(* IEC 61131-3 sources: elnaProjects/ElpcLogic/PomarKc7Changed/FunctionBlocks (part 6) *)

(* ---- ppuAlg.st ---- *)
FUNCTION_BLOCK ppuAlg

VAR_IN_OUT
	StrAlg : struct_Alg;
END_VAR

VAR
	BMP_Err : struct_PhaseAlgoritm;
	Level_masla_Norm : struct_PhaseAlgoritm;
	T_masla_Norm : struct_PhaseAlgoritm;
	Krans_ready_to_move : struct_PhaseAlgoritm;
END_VAR

VAR_IN_OUT
	Krans_Poloj : struct_PhaseAlgoritm;
	Net_AO_KC_SHKS04M : struct_PhaseAlgoritm;
	EGPA_Stop : struct_PhaseAlgoritm;
	Avt_SHU_vkl : struct_PhaseAlgoritm;
	All_IM_Off : struct_PhaseAlgoritm;
	Nalichie220_SHU_Ai : struct_PhaseAlgoritm;
	BP_Norm : struct_PhaseAlgoritm;
	Naprajenie_U_IM : struct_PhaseAlgoritm;
	MV_Poloj_RolledON : struct_PhaseAlgoritm;
	MV_Poloj_RolledOFF : struct_PhaseAlgoritm;
	NOTAnalogNS : struct_PhaseAlgoritm;
	Net_ASPS_Analogs : struct_PhaseAlgoritm;
	Not_AS : struct_PhaseAlgoritm;
	Gotov_Vozb : struct_PhaseAlgoritm;
	Reactornyi_P : struct_PhaseAlgoritm;
	Chastotnyi_P : struct_PhaseAlgoritm;
	dP_kr1 : struct_PhaseAlgoritm;
	Auto_Rej : struct_PhaseAlgoritm;
	CK_IM_Norm : struct_PhaseAlgoritm;
	HAnd_Mode : struct_PhaseAlgoritm;
	Impuls_Gaz : struct_PhaseAlgoritm;
END_VAR

VAR
	fb_BMP_Err : fb_ph_CustomPhase;
	fb_Level_masla_Norm : fb_ph_CustomPhase;
	fb_T_masla_Norm : fb_ph_CustomPhase;
	fb_Krans_ready_to_move : fb_ph_CustomPhase;
	fb_Krans_Poloj : fb_ph_CustomPhase;
	fb_Net_AO_KC_SHKS04M : fb_ph_CustomPhase;
	fb_EGPA_Stop : fb_ph_CustomPhase;
	fb_Avt_SHU_vkl : fb_ph_CustomPhase;
	fb_All_IM_Off : fb_ph_CustomPhase;
	fb_Nalichie220_SHU_Ai : fb_ph_CustomPhase;
	fb_BP_Norm : fb_ph_CustomPhase;
	fb_Naprajenie_U_IM : fb_ph_CustomPhase;
	fb_MV_Poloj_RolledON : fb_ph_CustomPhase;
	fb_MV_Poloj_RolledOFF : fb_ph_CustomPhase;
	fb_NOTAnalogNS : fb_ph_CustomPhase;
	fb_Net_ASPS_Analogs : fb_ph_CustomPhase;
	fb_Not_AS : fb_ph_CustomPhase;
	fb_Gotov_Vozb : fb_ph_CustomPhase;
	fb_Reactornyi_P : fb_ph_CustomPhase;
	fb_Chastotnyi_P : fb_ph_CustomPhase;
	fb_dP_kr1 : fb_ph_CustomPhase;
	fb_Auto_Rej : fb_ph_CustomPhase;
	fb_CK_IM_Norm : fb_ph_CustomPhase;
	fb_HAnd_Mode : fb_ph_CustomPhase;
	fb_Impuls_Gaz : fb_ph_CustomPhase;
	_sunpackerCommand : fb_sunpackerCommand;
	modeR_Trig : R_TRIG;
	modeF_Trig : F_TRIG;
	_statusAi : TYPE_StatusAi;
	_Answers : TYPE_Answers;
	_statusDualInput : TYPE_statusDualInput;
	_DualStateImAction : TYPE_DualStateImAction;
	_PhaseAlgoritmAction : TYPE_PhaseAlgoritmAction;
	_basketStats : TYPE_basketStats;
END_VAR

VAR_OUTPUT
	puskAllowed : BOOL;
	testAllowed : BOOL;
END_VAR

VAR
	ppuDone : BOOL;
	source : BYTE;
	cmd : BYTE;
	lastCmd : BYTE;
	source_for_Status : BYTE;
	cmd_for_Status : BYTE;
	command_error_for_Status : BYTE;
	resetCmdTimer : TON;
	resetCmdTimerPriznak : BOOL;
	onInit : BOOL;
END_VAR

VAR_EXTERNAL
	IM : ImConfig;
	ai : AiConfig;
	di : DiConfig;
	algManager : struct_AlgoritmsManager;
	protectManager : struct_ProtectionsManager;
	NotHasRezervNU : BOOL;
	ModeGpa : TYPE_ModeGpa;
	algoritms : AlgoritmsConfig;
END_VAR

IF NOT onInit THEN

    fb_BMP_Err(phaseNumber:=0);
    fb_Level_masla_Norm(phaseNumber:=1);
    fb_T_masla_Norm(phaseNumber:=2);
    fb_Krans_ready_to_move(phaseNumber:=5);
    fb_Krans_Poloj(phaseNumber:=6);
    fb_Net_AO_KC_SHKS04M(phaseNumber:=7);
    fb_EGPA_Stop(phaseNumber:=9);
    fb_Avt_SHU_vkl(phaseNumber:=10);
    fb_All_IM_Off(phaseNumber:=11);
    fb_Nalichie220_SHU_Ai(phaseNumber:=12);
    fb_BP_Norm(phaseNumber:=13);
    fb_Naprajenie_U_IM(phaseNumber:=14);
    fb_MV_Poloj_RolledON(phaseNumber:=15);
    fb_MV_Poloj_RolledOFF(phaseNumber:=16);
    fb_NOTAnalogNS(phaseNumber:=17);
    fb_Net_ASPS_Analogs(phaseNumber:=18);
    fb_Not_AS(phaseNumber:=19);
    fb_Gotov_Vozb(phaseNumber:=20);
    fb_Reactornyi_P(phaseNumber:=21);
    fb_Chastotnyi_P(phaseNumber:=22);
    fb_dP_kr1(phaseNumber:=23);
    fb_Auto_Rej(phaseNumber:=24);
    fb_CK_IM_Norm(phaseNumber:=25);
    fb_HAnd_Mode(phaseNumber:=26);
    fb_Impuls_Gaz(phaseNumber:=27);

onInit:=TRUE;
END_IF;

fb_BMP_Err(StrPh:=BMP_Err);
fb_Level_masla_Norm(StrPh:=Level_masla_Norm);
fb_T_masla_Norm(StrPh:=T_masla_Norm);
fb_Krans_ready_to_move(StrPh:=Krans_ready_to_move);
fb_Krans_Poloj(StrPh:=Krans_Poloj);
fb_Net_AO_KC_SHKS04M(StrPh:=Net_AO_KC_SHKS04M);
fb_EGPA_Stop(StrPh:=EGPA_Stop);
fb_Avt_SHU_vkl(StrPh:=Avt_SHU_vkl);
fb_All_IM_Off(StrPh:=All_IM_Off);
fb_Nalichie220_SHU_Ai(StrPh:=Nalichie220_SHU_Ai);
fb_BP_Norm(StrPh:=BP_Norm);
fb_Naprajenie_U_IM(StrPh:=Naprajenie_U_IM);
fb_MV_Poloj_RolledON(StrPh:=MV_Poloj_RolledON);
fb_MV_Poloj_RolledOFF(StrPh:=MV_Poloj_RolledOFF);
fb_NOTAnalogNS(StrPh:=NOTAnalogNS);
fb_Net_ASPS_Analogs(StrPh:=Net_ASPS_Analogs);
fb_Not_AS(StrPh:=Not_AS);
fb_Gotov_Vozb(StrPh:=Gotov_Vozb);
fb_Reactornyi_P(StrPh:=Reactornyi_P);
fb_Chastotnyi_P(StrPh:=Chastotnyi_P);
fb_dP_kr1(StrPh:=dP_kr1);
fb_Auto_Rej(StrPh:=Auto_Rej);
fb_CK_IM_Norm(StrPh:=CK_IM_Norm);
fb_HAnd_Mode(StrPh:=HAnd_Mode);
fb_Impuls_Gaz(StrPh:=Impuls_Gaz);

IF StrAlg.isRuning THEN

    (*BMP_Err.top:= ((BMPERR_k = 0) OR (kontroller.imit)); надо разобраться кто такой BMPERR_k*)
    (*уровень масла в норме*)
    Level_masla_Norm.top := (ai.Yroven_masla_MB.interval = _statusAi.normal);

    (*температура масла в норме*)
    T_masla_Norm.top:= (ai.Tmasla_MB.interval = _statusAi.normal);

    (*kраны готовы к управлению*)
    Krans_ready_to_move.top:= NOT (IM.Kran1.So OR IM.Kran1.Sz OR IM.Kran2.So OR IM.Kran2.Sz OR IM.Kran3.So OR
                                   IM.Kran3.Sz OR IM.Kran3b.So OR IM.Kran3b.Sz OR IM.Kran4.So OR IM.Kran4.Sz OR
			     IM.Kran5.So OR IM.Kran5.Sz OR IM.Kran6.So OR IM.Kran6.Sz);

    (*положение кранов верное*)
    Krans_Poloj.top:= (Im.Kran1.onStatus=_statusDualInput.STATUS_OFF) AND
		  (Im.Kran2.onStatus=_statusDualInput.STATUS_OFF) AND
		  (Im.Kran3.onStatus=_statusDualInput.STATUS_OFF) AND
		  (Im.Kran3b.onStatus=_statusDualInput.STATUS_ON) AND
		  (Im.Kran4.onStatus=_statusDualInput.STATUS_OFF) AND
		  (Im.Kran5.onStatus=_statusDualInput.STATUS_ON) AND
                      (Im.Kran6.onStatus=_statusDualInput.STATUS_ON);
    (*Нет АО от ШКС
    Net_AO_KC_SHKS04M.top:= haveAlarms(); кто такой haveAlarms*)

    (*Режим ЭГПА остановлен *)
    EGPA_Stop.top := (algManager.mode = ModeGpa.MODE_STOP);

    (*Автомат ШУ включен *)
    Avt_SHU_vkl.top := IM.SingleSignals.SHU_v_GPA_vkluch.Q;

    (*Все исполнительные механизмы выключены *)
    All_IM_Off.top := (IM.mv.onStatus=_statusDualInput.STATUS_OFF) AND (IM.pns.onStatus=_statusDualInput.STATUS_OFF) AND
                      (IM.nu1.onStatus=_statusDualInput.STATUS_OFF) AND (IM.nu2.onStatus=_statusDualInput.STATUS_OFF) AND
                      (IM.v1_Avom.onStatus=_statusDualInput.STATUS_OFF) AND (IM.v2_Avom.onStatus=_statusDualInput.STATUS_OFF) AND
		  (IM.v3_Avom.onStatus=_statusDualInput.STATUS_OFF)AND (IM.v4_Avom.onStatus=_statusDualInput.STATUS_OFF) AND
                      (IM.CMN.onStatus=_statusDualInput.STATUS_OFF) AND (IM.TEN_MB.onStatus=_statusDualInput.STATUS_OFF) AND
                      (IM.TEN_kollectora.onStatus=_statusDualInput.STATUS_OFF) AND (IM.KaloriferAVOM.onStatus=_statusDualInput.STATUS_OFF);

    (*Наличие 220 в шу*)
    Nalichie220_SHU_Ai.top :=	(ai.Kontrol_per_220V.interval = _statusAi.normal)	 AND (ai.Kontrol_post_220V.interval = _statusAi.normal);

    (*Блоки питания норм*)
    BP_Norm.top:=
		(IM.SingleSignals.Nalichie_BP1.Q AND
		IM.SingleSignals.Nalichie_BP2.Q AND
		IM.SingleSignals.Nalichie_BP3.Q AND
		IM.SingleSignals.Nalichie_BP4.Q AND
		IM.SingleSignals.Nalichie_BP5.Q AND
		IM.SingleSignals.Nalichie_BP6.Q AND
		IM.SingleSignals.Nalichie_BP7_BP8.Q AND
		IM.SingleSignals.Nalichie_BP9_BP10.Q AND

		IM.SingleSignals.Nalichie_220BEAO.Q AND
		IM.SingleSignals.Nalichie_per_220_na_vhode.Q AND
		IM.SingleSignals.Nalichie_post_220_na_vhode.Q AND
		IM.SingleSignals.Nalichie_BP11.Q AND
		IM.SingleSignals.Nalichie_BP12.Q);

    (*Напряжение исполнительниых механизмов
    Naprajenie_U_IM.top := IM.NalichieU_CMN.q AND IM.NalichieU_NU1.Q AND IM.Nalichie_CU_MV.Q  AND IM.NalichieU_NU2.Q AND
						IM.NalichieU_PNS.Q; нет сигналов таких *)

    (* положение тележки мв вкачена *)
    MV_Poloj_RolledON.top:= IM.mv.basketStatus = _basketStats.BASKET_ROLLEDIN;

    (* положение тележки мв выкачена *)
    MV_Poloj_RolledOFF.top:= IM.mv.basketStatus = _basketStats.BASKET_ROLLEDOUT;

    (* нет неисправных аналоговых сигналов *)
    NOTAnalogNS.top :=  NOT analogsNS();

    (* нет аварийных/предупредительных сигнализаций аналоговых сигналов *)
    Net_ASPS_Analogs.top := anyAnalogsPs(); (*Не понял где посмотреть наличие ас аналогов *)

    (* нет сработанных защит *)
    Not_AS.top := NOT anyProtectionSignaling();

    (* готовность возбудителя *)
    Gotov_Vozb.top:= IM.SingleSignals.Vozbud_gotovnost.Q;

    (* реакторный пуск *)
    Reactornyi_P.top := IM.SingleSignals.Reactorny_pusk.Q AND NOT IM.SingleSignals.Chastotny_pusk.Q;

    (* частотный пуск *)
    Chastotnyi_P.top:=IM.SingleSignals.Chastotny_pusk.Q AND NOT IM.SingleSignals.Reactorny_pusk.Q;

    (* нет перепада давления на кране 1 *)
    dP_kr1.top:= NOT IM.SingleSignals.dp_kran1_Less100.Q (*AND (IM.PerepadDavlenieKran1_CK.status = 1))*);

    (* в автоматическом ли режиме исполнительные механизмы *)
    (*Auto_Rej.top := im.NU1_Automat.Q AND im.PNS_Automat.Q AND im.NU2_Automat.Q;*)

    (* есть наряжение в цепях управления ИМ *)
    CK_IM_Norm.top := nsCepeiUpravlenya();

    (* ручной режим *)
    HAnd_Mode.top:= NOT im.SingleSignals.Rezhim_ruchnogo_regulirovaniya.Q;

    (* импульсный газ *)
    Impuls_Gaz.top:= ai.Pimpuls_gaz.interval=_statusAi.normal;

    ppuDone := BMP_Err.top AND
	     Level_masla_Norm.top AND
               T_masla_Norm.top AND
	     Krans_ready_to_move.top AND
	     Krans_Poloj.top AND
	     Net_AO_KC_SHKS04M.top AND
	     EGPA_Stop.top AND
               Avt_SHU_vkl.top AND
               All_IM_Off.top AND
               Nalichie220_SHU_Ai.top AND
               BP_Norm.top AND
               Naprajenie_U_IM.top AND
               MV_Poloj_RolledON.top AND
               MV_Poloj_RolledOFF.top AND
               NOTAnalogNS.top AND
               Net_ASPS_Analogs.top AND
               Not_AS.top AND
               Gotov_Vozb.top AND
               Reactornyi_P.top AND
               Chastotnyi_P.top AND
               dP_kr1.top AND
               Auto_Rej.top AND
               CK_IM_Norm.top AND
               HAnd_Mode.top AND
               Impuls_Gaz.top;

    puskAllowed:= ppuDone AND Im.mv.basketStatus = _basketStats.BASKET_ROLLEDIN;
    testAllowed:= ppuDone AND Im.mv.basketStatus = _basketStats.BASKET_ROLLEDOUT;

    modeR_Trig(CLK:=puskAllowed);
    modeF_Trig(CLK:=puskAllowed);

    IF modeR_Trig.Q THEN
	algManager.nMode:= ModeGpa.MODE_READY;
    END_IF;
    IF modeF_Trig.Q THEN
	algManager.nMode:= ModeGpa.MODE_STOP;
    END_IF;

    IF puskAllowed THEN
        algoritms.Apusk.inCanRun:= TRUE;
        algoritms.SemiAutoPusk.inCanRun:= TRUE;
    ELSE
        algoritms.Apusk.inCanRun:= FALSE;
        algoritms.SemiAutoPusk.inCanRun:= FALSE;
    END_IF;

    IF testAllowed THEN
        algoritms.testPms.inCanRun:=  TRUE;
        algoritms.testdPmg.inCanRun:= TRUE;
        algoritms.puskK.inCanRun:=    TRUE;
        algoritms.puskV.inCanRun:=    TRUE;
    ELSE
        algoritms.testPms.inCanRun:=  FALSE;
        algoritms.testdPmg.inCanRun:= FALSE;
        algoritms.puskK.inCanRun:=    FALSE;
        algoritms.puskV.inCanRun:=    FALSE;
    END_IF;

END_IF;

StrAlg.CanRun := StrAlg.inCanRun;
StrAlg.OpcCommandsDisabled := StrAlg.inOpcCommandsDisabled;

(* ---- Если управление с ВУ заблокировано, то  передаем команду из алгоритма ---- *)
IF StrAlg.inOpcCommandsDisabled THEN
	StrAlg.inCommand := StrAlg.inCommand_Alg;
ELSE (* иначе передаем команду с АРМа*)
	StrAlg.inCommand := StrAlg.inCommand_ARM;
END_IF;

_sunpackerCommand(command := StrAlg.inCommand);
	source := _sunpackerCommand.source;
	cmd := _sunpackerCommand.cmd;

IF cmd <> 0 AND lastCmd <> cmd AND (((NOT StrAlg.opcCommandsDisabled) AND source > 0) OR source = 0) then
	CASE BYTE_TO_INT(cmd) OF
		(*cmdRun*) 1: 	IF (StrAlg.CanRun) THEN
					StrAlg.isRuning := TRUE;
					StrAlg.isEnded := FALSE;
					StrAlg.hasError := FALSE;
					(*****************       OnRun       *****************)

					cmd_for_Status := cmd;
					source_for_Status := source;
					command_error_for_Status := 0;
				ELSE
					StrAlg.isRuning := FALSE;
					StrAlg.isEnded := FALSE;
					StrAlg.hasError 	:= FALSE;

					cmd_for_Status := 0;
					source_for_Status := source;
					command_error_for_Status := cmd;
				END_IF;
		(*cmdReset*) 2: 	StrAlg.isRuning := FALSE;
				StrAlg.isEnded := FALSE;
				StrAlg.hasError 	:= FALSE;

                                         (*****************       OnReset       *****************)

                                                  resetPhase(BMP_Err);
                                                  resetPhase(Level_masla_Norm);
                                                  resetPhase(T_masla_Norm);
                                                  resetPhase(Krans_ready_to_move);
                                                  resetPhase(Krans_Poloj);
                                                  resetPhase(Net_AO_KC_SHKS04M);
                                                  resetPhase(EGPA_Stop);
                                                  resetPhase(Avt_SHU_vkl);
                                                  resetPhase(All_IM_Off);
                                                  resetPhase(Nalichie220_SHU_Ai);
                                                  resetPhase(BP_Norm);
                                                  resetPhase(Naprajenie_U_IM);
                                                  resetPhase(MV_Poloj_RolledON);
                                                  resetPhase(MV_Poloj_RolledOFF);
                                                  resetPhase(NOTAnalogNS);
                                                  resetPhase(Net_ASPS_Analogs);
                                                  resetPhase(Not_AS);
                                                  resetPhase(Gotov_Vozb);
                                                  resetPhase(Reactornyi_P);
                                                  resetPhase(Chastotnyi_P);
                                                  resetPhase(dP_kr1);
                                                  resetPhase(Auto_Rej);
                                                  resetPhase(CK_IM_Norm);
                                                  resetPhase(HAnd_Mode);
                                                  resetPhase(Impuls_Gaz);

                                                  algoritms.testPms.inCanRun:=  FALSE;
                                                  algoritms.testdPmg.inCanRun:= FALSE;
                                                  algoritms.puskK.inCanRun:=    FALSE;
                                                  algoritms.puskV.inCanRun:=    FALSE;

                                        StrAlg.inCanRun:=FALSE;
                                        puskAllowed:=FALSE;
                                        testAllowed:=FALSE;
                                        modeR_Trig(CLK:=FALSE);
                                        modeF_Trig(CLK:=FALSE);

				cmd_for_Status := cmd;
				source_for_Status := source;
				command_error_for_Status := 0;
	END_CASE;
	resetCmdTimer(IN := false);
	resetCmdTimerPriznak := TRUE;
END_IF;
lastCmd := cmd;

resetCmdTimer(IN := resetCmdTimerPriznak, PT := T#5S);
IF resetCmdTimer.Q THEN
	resetCmdTimerPriznak := FALSE;
	source_for_Status := 0;
	cmd_for_Status := 0;
	command_error_for_Status := 0;
END_IF;

StrAlg.Start:= BMP_Err.startStatus
            OR Level_masla_Norm.startStatus
            OR T_masla_Norm.startStatus
            OR Krans_ready_to_move.startStatus
            OR Krans_Poloj.startStatus
            OR Net_AO_KC_SHKS04M.startStatus
            OR EGPA_Stop.startStatus
            OR Avt_SHU_vkl.startStatus
            OR All_IM_Off.startStatus
            OR Nalichie220_SHU_Ai.startStatus
            OR BP_Norm.startStatus
            OR Naprajenie_U_IM.startStatus
            OR MV_Poloj_RolledON.startStatus
            OR MV_Poloj_RolledOFF.startStatus
            OR NOTAnalogNS.startStatus
            OR Net_ASPS_Analogs.startStatus
            OR Not_AS.startStatus
            OR Gotov_Vozb.startStatus
            OR Reactornyi_P.startStatus
            OR Chastotnyi_P.startStatus
            OR dP_kr1.startStatus
            OR Auto_Rej.startStatus
            OR CK_IM_Norm.startStatus
            OR HAnd_Mode.startStatus
            OR Impuls_Gaz.startStatus;

StrAlg.Error:= BMP_Err.errorStatus
            OR Level_masla_Norm.errorStatus
            OR T_masla_Norm.errorStatus
            OR Krans_ready_to_move.errorStatus
            OR Krans_Poloj.errorStatus
            OR Net_AO_KC_SHKS04M.errorStatus
            OR EGPA_Stop.errorStatus
            OR Avt_SHU_vkl.errorStatus
            OR All_IM_Off.errorStatus
            OR Nalichie220_SHU_Ai.errorStatus
            OR BP_Norm.errorStatus
            OR Naprajenie_U_IM.errorStatus
            OR MV_Poloj_RolledON.errorStatus
            OR MV_Poloj_RolledOFF.errorStatus
            OR NOTAnalogNS.errorStatus
            OR Net_ASPS_Analogs.errorStatus
            OR Not_AS.errorStatus
            OR Gotov_Vozb.errorStatus
            OR Reactornyi_P.errorStatus
            OR Chastotnyi_P.errorStatus
            OR dP_kr1.errorStatus
            OR Auto_Rej.errorStatus
            OR CK_IM_Norm.errorStatus
            OR HAnd_Mode.errorStatus
            OR Impuls_Gaz.errorStatus;

StrAlg.Top:=   BMP_Err.topStatus
            OR Level_masla_Norm.topStatus
            OR T_masla_Norm.topStatus
            OR Krans_ready_to_move.topStatus
            OR Krans_Poloj.topStatus
            OR Net_AO_KC_SHKS04M.topStatus
            OR EGPA_Stop.topStatus
            OR Avt_SHU_vkl.topStatus
            OR All_IM_Off.topStatus
            OR Nalichie220_SHU_Ai.topStatus
            OR BP_Norm.topStatus
            OR Naprajenie_U_IM.topStatus
            OR MV_Poloj_RolledON.topStatus
            OR MV_Poloj_RolledOFF.topStatus
            OR NOTAnalogNS.topStatus
            OR Net_ASPS_Analogs.topStatus
            OR Not_AS.topStatus
            OR Gotov_Vozb.topStatus
            OR Reactornyi_P.topStatus
            OR Chastotnyi_P.topStatus
            OR dP_kr1.topStatus
            OR Auto_Rej.topStatus
            OR CK_IM_Norm.topStatus
            OR HAnd_Mode.topStatus
            OR Impuls_Gaz.topStatus;

(*TODO: TYPE PROGRAM CODE HERE*)
StrAlg.status :=  SHL(BYTE_TO_DWORD(source_for_Status), 29)
			OR SHL(BYTE_TO_DWORD(cmd_for_Status), 26)
			OR SHL(BYTE_TO_DWORD(command_error_for_Status), 23)
			OR SHL(BOOL_TO_DWORD(StrAlg.OpcCommandsDisabled ), 21)
                              OR SHL(BOOL_TO_DWORD(testAllowed),16)
                              OR SHL(BOOL_TO_DWORD(puskAllowed),15)
			OR SHL(BOOL_TO_DWORD(StrAlg.hasError),4)
			OR SHL(BOOL_TO_DWORD(StrAlg.CanRun),2)
			OR SHL(BOOL_TO_DWORD(StrAlg.isEnded),1)
			OR BOOL_TO_DWORD(StrAlg.isRuning);

(* ---- proc_AI.st ---- *)
FUNCTION_BLOCK proc_AI

VAR
	fb_TStalisStatoraKanal1 : fb_AiSourceMlp; (*[A1-14:1, AI0] Резерв*)
	fb_TStalisStatoraKanal2 : fb_AiSourceMlp; (*[A1-14:2, AI1] Резерв*)
	fb_TStalisStatoraKanal3 : fb_AiSourceMlp; (*[A1-14:3, AI2] Резерв*)
	fb_TMediStatoraKanal1 : fb_AiSourceMlp; (*[A1-14:4, AI3] Резерв*)
	fb_TMediStatoraKanal2 : fb_AiSourceMlp; (*[A1-14:5, AI4] Резерв*)
	fb_TMediStatoraKanal3 : fb_AiSourceMlp; (*[A1-14:6, AI5] Резерв*)
	fb_TOpornogoPodshipnikaEDT_1 : fb_AiSourceMlp; (*[A1-14:7, AI6] Резерв*)
	fb_TOpornoYpornogoPodshipnikaEDT_2 : fb_AiSourceMlp; (*[A1-14:8, AI7] Резерв*)
	fb_TOpornoYpornogoPodshipnikaKolesaRedEDT_3 : fb_AiSourceMlp;
	fb_TOpornoYpornogoPodshipnikaKolesaRedHT_4 : fb_AiSourceMlp;
	fb_TOpornogoPodshipnikaShesterniReduktoraT_5 : fb_AiSourceMlp;
	fb_TOpornogoPodshipnikaReduktoraHT_6 : fb_AiSourceMlp;
	fb_TOpornoYpornogoPodshipnikaNagnetateljaT_7_1 : fb_AiSourceMlp;
	fb_TOpornoYpornogoPodshipnikaNagnetateljaT_7_2 : fb_AiSourceMlp;
	fb_TOpornoYpornogoPodshipnikaSvobodnogoKoncaNT_8_1 : fb_AiSourceMlp;
	fb_TOpornoYpornogoPodshipnikaSvobodnogoKoncaNT_8_2 : fb_AiSourceMlp;
	fb_TYpornogoPodshipnikaRabKolodokHT_9_1 : fb_AiSourceMlp;
	fb_TYpornogoPodshipnikaRabKolodokHT_9_2 : fb_AiSourceMlp;
	fb_TYpornogoPodshipnikYstanKolodokHT_10_1 : fb_AiSourceMlp;
	fb_TYpornogoPodshipnikYstanKolodokHT_10_2 : fb_AiSourceMlp;
	fb_THolodnogoVozduhaEDKanall : fb_AiSourceMlp;
	fb_THolodnogoVozduhaEDKanal2 : fb_AiSourceMlp;
	fb_TGorjachegoVozduhaEDKanall : fb_AiSourceMlp;
	fb_TGorjachegoVozduhaEDKanal2 : fb_AiSourceMlp;
	fb_TNArujnogoVozduha : fb_AiSourceMlp;
	fb_TgazaNaVhodeH : fb_AiSourceMlp_timer;
	fb_TgazaNaVyhodeH : fb_AiSourceMlp;
	fb_TMasladoAVOM : fb_AiSourceMlp;
	fb_TMaslaPosleAVOM : fb_AiSourceMlp;
	fb_TMaslaMB : fb_AiSourceMlp;
	fb_TEmperatura_v_SHU : fb_AiSourceMlp_timer;
	fb_DavlenijaMasloSmNizkoe : fb_AiSourceMlp;
	fb_PerepadDavlenieNaMasloFiltre : fb_AiSourceMlp;
	fb_DavlenijaMasloSmVysokoe : fb_AiSourceMlp;
	fb_DavlenijaMaslaPosleGNS : fb_AiSourceMlp;
	fb_DavlenijaMaslaPosleNU : fb_AiSourceMlp;
	fb_PerepadDavlenieNaKonfuzore : fb_AiSourceMlp;
	fb_OsSdvigNagnetatelja_Plus : fb_AiSourceMlp;
	fb_OsSdvigNagnetatelja_Minus : fb_AiSourceMlp;
	fb_PerepadDavlenieMasloGaz : fb_AiSourceMlp;
	fb_VibroSkorostOYPKolesaED_T3 : fb_AiSourceMlp;
	fb_DGazaNaVhodeNagnetatelja : fb_AiSourceMlp;
	fb_DGazaNaVyhodeNagnetatelja : fb_AiSourceMlp;
	fb_DavlenieImpulsGaz : fb_AiSourceMlp;
	fb_YrovenMaslaMB : fb_AiSourceMlp;
	fb_Kontrol_per220V : fb_AiSourceMlp;
	fb_Kontrol_post220V : fb_AiSourceMlp;
	fb_TMaslaMB_TEN : fb_AiSourceMlp;
	fb_VibroSkorostOPED_T1 : fb_AiSourceMlp;
	fb_VibroSkorostOYPED_T2 : fb_AiSourceMlp;
	fb_VibroSkorostOPKolesaRH_T4 : fb_AiSourceMlp;
	fb_VibroSkorostOPShesterniRED_T5 : fb_AiSourceMlp;
	fb_VibroSkorostOPShesterniReduktoraH_T6 : fb_AiSourceMlp;
	fb_TokStatora : fb_AiSourceMlp;
END_VAR

VAR_EXTERNAL
	arAIN_0 : TItemAIN;
	arAIN_1 : TItemAIN;
	arAIN_2 : TItemAIN;
	arAIN_3 : TItemAIN;
	arAIN_4 : TItemAIN;
	arAIN_5 : TItemAIN;
	arAIN_6 : TItemAIN;
	arAIN_7 : TItemAIN;
	arAIN_8 : TItemAIN;
	arAIN_9 : TItemAIN;
	arAIN_10 : TItemAIN;
	arAIN_11 : TItemAIN;
	arAIN_12 : TItemAIN;
	arAIN_13 : TItemAIN;
	arAIN_14 : TItemAIN;
	arAIN_15 : TItemAIN;
	ai : AiConfig;
	arAIN_16 : TItemAIN;
	arAIN_17 : TItemAIN;
	arAIN_18 : TItemAIN;
	arAIN_19 : TItemAIN;
	arAIN_20 : TItemAIN;
	arAIN_21 : TItemAIN;
	arAIN_22 : TItemAIN;
	arAIN_23 : TItemAIN;
	arAIN_24 : TItemAIN;
	arAIN_25 : TItemAIN;
	arAIN_26 : TItemAIN;
	arAIN_27 : TItemAIN;
	arAIN_28 : TItemAIN;
	arAIN_29 : TItemAIN;
	arAIN_30 : TItemAIN;
	arAIN_31 : TItemAIN;
	arAIN_32 : TItemAIN;
	arAIN_33 : TItemAIN;
	arAIN_34 : TItemAIN;
	arAIN_35 : TItemAIN;
	arAIN_36 : TItemAIN;
	arAIN_37 : TItemAIN;
	arAIN_38 : TItemAIN;
	arAIN_39 : TItemAIN;
	arAIN_40 : TItemAIN;
	arAIN_41 : TItemAIN;
	arAIN_42 : TItemAIN;
	arAIN_43 : TItemAIN;
	arAIN_44 : TItemAIN;
	arAIN_45 : TItemAIN;
	arAIN_46 : TItemAIN;
	arAIN_47 : TItemAIN;
	arAIN_48 : TItemAIN;
	arAIN_49 : TItemAIN;
	arAIN_50 : TItemAIN;
	arAIN_51 : TItemAIN;
	arAIN_52 : TItemAIN;
	arAIN_53 : TItemAIN;
	arAIN_54 : TItemAIN;
	arAIN_55 : TItemAIN;
	arAIN_56 : TItemAIN;
	arAIN_57 : TItemAIN;
	arAIN_58 : TItemAIN;
	arAIN_59 : TItemAIN;
	arAIN_60 : TItemAIN;
	arAIN_61 : TItemAIN;
	arAIN_62 : TItemAIN;
	arAIN_63 : TItemAIN;
	arAIN_64 : TItemAIN;
	arAIN_65 : TItemAIN;
	arERR_3 : TItemDIN;
	arERR_4 : TItemDIN;
	arERR_5 : TItemDIN;
	arERR_6 : TItemDIN;
	arERR_7 : TItemDIN;
	arERR_8 : TItemDIN;
	arERR_9 : TItemDIN;
	A1_10_err_mode : UINT;
	A1_11_err_mode : UINT;
	A1_4_err_mode : UINT;
	A1_5_err_mode : UINT;
	A1_6_err_mode : UINT;
	A1_7_err_mode : UINT;
	A1_8_err_mode : UINT;
	A1_9_err_mode : UINT;
	A2_2_err_mode : UINT;
	A2_3_err_mode : UINT;
	AI_0_dblValue : LREAL;
	AI_10_dblValue : LREAL;
	AI_11_dblValue : LREAL;
	AI_12_dblValue : LREAL;
	AI_13_dblValue : LREAL;
	AI_14_dblValue : LREAL;
	AI_15_dblValue : LREAL;
	AI_16_dblValue : LREAL;
	AI_17_dblValue : LREAL;
	AI_18_dblValue : LREAL;
	AI_19_dblValue : LREAL;
	AI_1_dblValue : LREAL;
	AI_20_dblValue : LREAL;
	AI_21_dblValue : LREAL;
	AI_22_dblValue : LREAL;
	AI_23_dblValue : LREAL;
	AI_24_dblValue : LREAL;
	AI_25_dblValue : LREAL;
	AI_26_dblValue : LREAL;
	AI_27_dblValue : LREAL;
	AI_28_dblValue : LREAL;
	AI_29_dblValue : LREAL;
	AI_2_dblValue : LREAL;
	AI_30_dblValue : LREAL;
	AI_31_dblValue : LREAL;
	AI_32_dblValue : LREAL;
	AI_33_dblValue : LREAL;
	AI_34_dblValue : LREAL;
	AI_35_dblValue : LREAL;
	AI_36_dblValue : LREAL;
	AI_37_dblValue : LREAL;
	AI_38_dblValue : LREAL;
	AI_39_dblValue : LREAL;
	AI_3_dblValue : LREAL;
	AI_40_dblValue : LREAL;
	AI_41_dblValue : LREAL;
	AI_42_dblValue : LREAL;
	AI_43_dblValue : LREAL;
	AI_44_dblValue : LREAL;
	AI_45_dblValue : LREAL;
	AI_46_dblValue : LREAL;
	AI_47_dblValue : LREAL;
	AI_48_dblValue : LREAL;
	AI_49_dblValue : LREAL;
	AI_4_dblValue : LREAL;
	AI_50_dblValue : LREAL;
	AI_51_dblValue : LREAL;
	AI_52_dblValue : LREAL;
	AI_53_dblValue : LREAL;
	AI_54_dblValue : LREAL;
	AI_55_dblValue : LREAL;
	AI_56_dblValue : LREAL;
	AI_57_dblValue : LREAL;
	AI_58_dblValue : LREAL;
	AI_59_dblValue : LREAL;
	AI_5_dblValue : LREAL;
	AI_60_dblValue : LREAL;
	AI_61_dblValue : LREAL;
	AI_62_dblValue : LREAL;
	AI_63_dblValue : LREAL;
	AI_64_dblValue : LREAL;
	AI_65_dblValue : LREAL;
	AI_66_dblValue : LREAL;
	AI_67_dblValue : LREAL;
	AI_68_dblValue : LREAL;
	AI_69_dblValue : LREAL;
	AI_6_dblValue : LREAL;
	AI_70_dblValue : LREAL;
	AI_71_dblValue : LREAL;
	AI_72_dblValue : LREAL;
	AI_73_dblValue : LREAL;
	AI_74_dblValue : LREAL;
	AI_75_dblValue : LREAL;
	AI_76_dblValue : LREAL;
	AI_77_dblValue : LREAL;
	AI_78_dblValue : LREAL;
	AI_79_dblValue : LREAL;
	AI_7_dblValue : LREAL;
	AI_8_dblValue : LREAL;
	AI_9_dblValue : LREAL;
END_VAR

(* Циклический опрос. Входные аналоговые параметры *)

(* [A1-9, AI5-4]  dР газа на конфузоре *)
fb_PerepadDavlenieNaKonfuzore(arAIN := arAIN_40, strAI := ai.dPgaza_na_konfuzore, err_mod:=arERR_8);
AI_40_dblValue := arAIN_40.dblValue;

(* [A1-9, AI5-0] dР масла на масляном фильтре *)
fb_PerepadDavlenieNaMasloFiltre(arAIN := arAIN_34, strAI := ai.dPgaza_na_maslo_filtre, err_mod:=arERR_8);
AI_34_dblValue := arAIN_34.dblValue;

(* [A1-9, AI5-7]  dР масло-газ *)
fb_PerepadDavlenieMasloGaz(arAIN := arAIN_41, strAI := ai.dPmaslo_gaz, err_mod:=arERR_8);
AI_41_dblValue := arAIN_41.dblValue;

(* [A1-10, AI6-2] Р газа на входе нагнетателя *)
fb_DGazaNaVhodeNagnetatelja(arAIN := arAIN_44, strAI := ai.Pgaza_na_vhode_nagnetatelia, err_mod:=arERR_9);
AI_44_dblValue := arAIN_44.dblValue;

(* [A1-10, AI6-3] Р газа на выходе нагнетателя *)
fb_DGazaNaVyhodeNagnetatelja(arAIN := arAIN_45, strAI := ai.Pgaza_na_vyhode_nagnetatelia, err_mod:=arERR_9);
AI_45_dblValue := arAIN_45.dblValue;

(* [A1-9, AI5-3]  Р масла после НУ *)
fb_DavlenijaMaslaPosleNU(arAIN := arAIN_37, strAI := ai.Pmasla_posle_NU, err_mod:=arERR_8);
AI_37_dblValue := arAIN_37.dblValue;

(* [A1-8, AI4-6]  Р масла смазки низкое) *)
fb_DavlenijaMasloSmNizkoe(arAIN := arAIN_33, strAI := ai.Pmaslo_sm_nizkoe, err_mod:=arERR_7);
AI_33_dblValue := arAIN_33.dblValue;

(* [A1-9, AI5-2]  Р масла смазки после ГМНС *)
fb_DavlenijaMaslaPosleGNS(arAIN := arAIN_36, strAI := ai.Pmasla_posle_GNS, err_mod:=arERR_8);
AI_36_dblValue := arAIN_36.dblValue;

(* [A1-9, AI5-1]  Р масла смазки высокое *)
fb_DavlenijaMasloSmVysokoe(arAIN := arAIN_35, strAI := ai.Pmaslo_sm_vysokoe, err_mod:=arERR_8);
AI_35_dblValue := arAIN_35.dblValue;

(* [A1-7, AI3-2] Т наружного воздуха *)
fb_TNArujnogoVozduha(arAIN := arAIN_24, strAI := ai.Tnarujnogo_vozduha, err_mod:=arERR_6);
AI_24_dblValue := arAIN_24.dblValue;

(* [A1-8, AI4-0]  Т газа на входе нагнетателя *)
fb_TgazaNaVhodeH(arAIN := arAIN_25, strAI := ai.Tgaza_na_vhode_H, err_mod:=arERR_7);
AI_25_dblValue := arAIN_25.dblValue;

(* [A1-8, AI4-1] Т газа на выходе нагнетателя *)
fb_TgazaNaVyhodeH(arAIN := arAIN_26, strAI := ai.Tgaza_na_vyhode_H, err_mod:=arERR_7);
AI_26_dblValue := arAIN_26.dblValue;

(* [A1-6, AI2-7]  Т горячего воздуха в ЭД, точка 1 *)
fb_TGorjachegoVozduhaEDKanall(arAIN := arAIN_22, strAI := ai.Tgorjachego_vozduha_ED_kanal_1, err_mod:=arERR_5);
AI_22_dblValue := arAIN_22.dblValue;

(* [A1-7, AI3-0] Т горячего воздуха в ЭД, точка 2 *)
fb_TGorjachegoVozduhaEDKanal2(arAIN := arAIN_23, strAI := ai.Tgorjachego_vozduha_ED_kanal_2, err_mod:=arERR_6);
AI_23_dblValue := arAIN_23.dblValue;

(* [A1-8, AI4-4] Т масла в маслобаке *)
fb_TMaslaMB(arAIN := arAIN_29, strAI := ai.Tmasla_MB, err_mod:=arERR_7);
AI_29_dblValue := arAIN_29.dblValue;

(* [A1-8, AI4-4] Т масла в маслобаке над ТЭНом *)
fb_TMaslaMB_TEN(arAIN := arAIN_30, strAI := ai.Tmasla_MB_TEN, err_mod:=arERR_7);
AI_30_dblValue := arAIN_30.dblValue;

(* [A1-8, AI4-2] Т масла до АВО М *)
fb_TMasladoAVOM(arAIN := arAIN_27, strAI := ai.Tgorjachego_vozduha_ED_kanal_2, err_mod:=arERR_7);
AI_27_dblValue := arAIN_27.dblValue;

(* [A1-8, AI4-3] Т масла после АВО М *)
fb_TMaslaPosleAVOM(arAIN := arAIN_28, strAI := ai.Tmasla_posle_AVOM, err_mod:=arERR_7);
AI_28_dblValue := arAIN_28.dblValue;

(* [A1-4, AI0-3] Т Т меди статора фаза 1 *)
fb_TMediStatoraKanal1(arAIN := arAIN_3, strAI := ai.Tmedi_statora_kanal_1, err_mod:=arERR_3);
AI_3_dblValue := arAIN_3.dblValue;

(* [A1-4, AI0-4] Т обмотки фазы 3 канал *)
fb_TMediStatoraKanal2(arAIN := arAIN_4, strAI := ai.Tmedi_statora_kanal_2, err_mod:=arERR_3);
AI_4_dblValue := arAIN_4.dblValue;

(* [A1-4, AI0-5] Т меди статора фаза 2 *)
fb_TMediStatoraKanal3(arAIN := arAIN_5, strAI := ai.Tmedi_statora_kanal_3, err_mod:=arERR_3);
AI_5_dblValue := arAIN_5.dblValue;

(* [A1-4, AI0-6] Т ОП ЭД со стороны свободного конца (т.1) } *)
fb_TOpornogoPodshipnikaEDT_1(arAIN := arAIN_6, strAI := ai.Toporno_podshipnika_EDT_1, err_mod:=arERR_3);
AI_6_dblValue := arAIN_6.dblValue;

(* [A1-5, AI1-0]  Т ОУП ЭД со стороны редуктора (т.2) *)
fb_TOpornoYpornogoPodshipnikaEDT_2(arAIN := arAIN_7, strAI := ai.Toy_podshipnika_EDT_2, err_mod:=arERR_4);
AI_7_dblValue := arAIN_7.dblValue;

(* [A1-5, AI1-1]  Т ОУП колеса редуктора со стороны ЭД (т.3) *)
fb_TOpornoYpornogoPodshipnikaKolesaRedEDT_3(arAIN := arAIN_8, strAI := ai.Toy_podshipnika_kol_EDT_3, err_mod:=arERR_4);
AI_8_dblValue := arAIN_8.dblValue;

(* [A1-5, AI1-2]Т ОП колеса редуктора со стороны Н (т.4) *)
fb_TOpornoYpornogoPodshipnikaKolesaRedHT_4(arAIN := arAIN_9, strAI := ai.Toy_podshipnika_kol_EDT_4, err_mod:=arERR_4);
AI_9_dblValue := arAIN_9.dblValue;

(* [A1-5, AI1-3] Т ОП шестерни редуктора со стороны ЭД (т.5) *)
fb_TOpornogoPodshipnikaShesterniReduktoraT_5(arAIN := arAIN_10, strAI := ai.Toy_podshipnika_shest_red_EDT_5, err_mod:=arERR_4);
AI_10_dblValue := arAIN_10.dblValue;

(* [A1-5, AI1-4]  Т ОП шестерни редуктора со стороны Н (т.6) *)
fb_TOpornogoPodshipnikaReduktoraHT_6(arAIN := arAIN_11, strAI := ai.Ty_podshipnika_red_EDT_6, err_mod:=arERR_4);
AI_11_dblValue := arAIN_11.dblValue;

(* [A1-5, AI1-5]  Т ОП Н со стороны редуктора (т.7) *)
fb_TOpornoYpornogoPodshipnikaNagnetateljaT_7_1(arAIN := arAIN_12, strAI := ai.Ty_podshipnika_nagnet_EDT_7_1, err_mod:=arERR_4);
AI_12_dblValue := arAIN_12.dblValue;

(* [A1-5, AI1-5]  Т ОП Н со стороны редуктора (т.7) *)
fb_TOpornoYpornogoPodshipnikaNagnetateljaT_7_2(arAIN := arAIN_13, strAI := ai.Ty_podshipnika_nagnet_EDT_7_2, err_mod:=arERR_4);
AI_13_dblValue := arAIN_13.dblValue;

(* [A1-5, AI1-7]  Т ОП Н со стороны свободного вала (т.8) *)
fb_TOpornoYpornogoPodshipnikaSvobodnogoKoncaNT_8_1(arAIN := arAIN_14, strAI := ai.Toy_podshipnika_svobod_konca_EDT_8_1, err_mod:=arERR_4);
AI_14_dblValue := arAIN_14.dblValue;

(* [A1-5, AI1-7]  Т ОП Н со стороны свободного вала (т.8) *)
fb_TOpornoYpornogoPodshipnikaSvobodnogoKoncaNT_8_2(arAIN := arAIN_15, strAI := ai.Toy_podshipnika_svobod_konca_EDT_8_2, err_mod:=arERR_4);
AI_15_dblValue := arAIN_15.dblValue;

(* [A1-6, AI2-1]  Т УП рабочих колодок нагнетателя(т9) *)
fb_TYpornogoPodshipnikaRabKolodokHT_9_1(arAIN := arAIN_16, strAI := ai.Toy_podshipnika_rab_kol_EDT_9_1, err_mod:=arERR_5);
AI_16_dblValue := arAIN_16.dblValue;

(* [A1-6, AI2-1]  Т УП рабочих колодок нагнетателя(т9) *)
fb_TYpornogoPodshipnikaRabKolodokHT_9_2(arAIN := arAIN_17, strAI := ai.Toy_podshipnika_rab_kol_EDT_9_2, err_mod:=arERR_5);
AI_17_dblValue := arAIN_17.dblValue;

(* [A1-6, AI2-3]  Т ОП установочных колодок нагнетателя(т10) *)
fb_TYpornogoPodshipnikYstanKolodokHT_10_1(arAIN := arAIN_18, strAI := ai.Toy_podshipnika_nerab_kol_EDT_10_1, err_mod:=arERR_5);
AI_18_dblValue := arAIN_18.dblValue;

(* [A1-6, AI2-3]  Т ОП установочных колодок нагнетателя(т10) *)
fb_TYpornogoPodshipnikYstanKolodokHT_10_2(arAIN := arAIN_19, strAI := ai.Toy_podshipnika_nerab_kol_EDT_10_2, err_mod:=arERR_5);
AI_19_dblValue := arAIN_19.dblValue;

(* [A1-4, AI0-0] Т стали статора фаза 1 *)
fb_TStalisStatoraKanal1(arAIN := arAIN_0, strAI := ai.Tstali_statora_kanal_1, err_mod:=arERR_3);
AI_0_dblValue := arAIN_0.dblValue;

(* [A1-4, AI0-1] Т стали статора фаза 2 *)
fb_TStalisStatoraKanal2(arAIN := arAIN_1, strAI := ai.Tstali_statora_kanal_2, err_mod:=arERR_3);
AI_1_dblValue := arAIN_1.dblValue;

(* [A1-4, AI0-2] Т стали статора фаза 3 *)
fb_TStalisStatoraKanal3(arAIN := arAIN_2, strAI := ai.Tstali_statora_kanal_3, err_mod:=arERR_3);
AI_2_dblValue := arAIN_2.dblValue;

(* [A1-6, AI2-5] Т холодного воздуха в ЭД, точка 1 *)
fb_THolodnogoVozduhaEDKanall(arAIN := arAIN_20, strAI := ai.Tholodnogo_vozduha_ED_kanal_1, err_mod:=arERR_5);
AI_20_dblValue := arAIN_20.dblValue;

(* [A1-6, AI2-6] Т холодного воздуха в ЭД, точка 2 *)
fb_THolodnogoVozduhaEDKanal2(arAIN := arAIN_21, strAI := ai.Tholodnogo_vozduha_ED_kanal_2, err_mod:=arERR_5);
AI_21_dblValue := arAIN_21.dblValue;

(* [A1-10, AI6-5] Уровень масла в маслобаке *)
fb_YrovenMaslaMB(arAIN := arAIN_48, strAI := ai.Yroven_masla_MB, err_mod:=arERR_9);
AI_48_dblValue := arAIN_48.dblValue;

(* [A1-10, AI6-5] Уровень масла в маслобаке *)
fb_VibroSkorostOPED_T1(arAIN := arAIN_56, strAI := ai.Kontrol_post_220V, err_mod:=arERR_9);
AI_56_dblValue := arAIN_56.dblValue;

(* [A1-10, AI6-5] Уровень масла в маслобаке *)
fb_VibroSkorostOYPED_T2(arAIN := arAIN_57, strAI := ai.Vibro_skorost_OPED_T1, err_mod:=arERR_9);
AI_57_dblValue := arAIN_57.dblValue;

(* [A1-10, AI6-5] Уровень масла в маслобаке *)
fb_VibroSkorostOPKolesaRH_T4(arAIN := arAIN_59, strAI := ai.Vibro_skorost_OP_kolesa_RH_T4, err_mod:=arERR_9);
AI_59_dblValue := arAIN_59.dblValue;

(* [A1-10, AI6-5] Уровень масла в маслобаке *)
fb_VibroSkorostOPShesterniRED_T5(arAIN := arAIN_60, strAI := ai.Vibro_skorost_OP_shesterni_RED_T5, err_mod:=arERR_9);
AI_60_dblValue := arAIN_60.dblValue;

(* [A1-10, AI6-5] Уровень масла в маслобаке *)
fb_VibroSkorostOPShesterniReduktoraH_T6(arAIN := arAIN_61, strAI := ai.Vibro_skorost_OP_shesterni_RED_T6, err_mod:=arERR_9);
AI_61_dblValue := arAIN_61.dblValue;

(**********************************************s Модуль A1-5 *********************************************************)
A1_4_err_mode := arERR_3.wValue;
A1_6_err_mode := arERR_5.wValue;
A1_5_err_mode := arERR_4.wValue;
A1_7_err_mode := arERR_6.wValue;

(********************************************** Модуль A1-8 *********************************************************)
(* [A1-8, AI4-5]  Температура в шкафу САУ *)
fb_TEmperatura_v_SHU(arAIN := arAIN_32, strAI := ai.Tshu, err_mod:=arERR_7);
AI_32_dblValue := arAIN_32.dblValue;

(* [A1-9, AI5-5]  Вибрация ротора нагнетателя т.4 *)
fb_OsSdvigNagnetatelja_Plus(arAIN := arAIN_42, strAI := ai.Os_sdvig_nagnetatelja_plus, err_mod:=arERR_8);
AI_42_dblValue := arAIN_42.dblValue;

(* [A1-9, AI5-6]  Осевой сдвиг ротора нагнетателя *)
fb_OsSdvigNagnetatelja_Minus(arAIN := arAIN_43, strAI := ai.Os_sdvig_nagnetatelja_minus, err_mod:=arERR_8);
AI_43_dblValue := arAIN_43.dblValue;

A1_9_err_mode := arERR_8.wValue;

(********************************************** Модуль A1-10 *********************************************************)
(* [A1-10, AI6-0] Температура внутри шкафа *)
fb_VibroSkorostOYPKolesaED_T3(arAIN := arAIN_58, strAI := ai.Vibro_skorost_OYP_kolesa_ED_T3, err_mod:=arERR_9);
AI_58_dblValue := arAIN_58.dblValue;

(* [A1-10, AI6-4] Активная мощность *)
fb_DavlenieImpulsGaz(arAIN := arAIN_46, strAI := ai.Pimpuls_gaz, err_mod:=arERR_9);
AI_46_dblValue := arAIN_46.dblValue;

(* [A1-10, AI6-6]  Напряжение питания ШУ, основной ввод *)
fb_Kontrol_per220V(arAIN := arAIN_52, strAI := ai.Kontrol_per_220V, err_mod:=arERR_9);
AI_52_dblValue := arAIN_52.dblValue;

(* [A1-10, AI6-7]  Напряжение питания ШУ, резервный ввод *)
fb_Kontrol_post220V(arAIN := arAIN_53, strAI := ai.Kontrol_post_220V, err_mod:=arERR_9);
AI_53_dblValue := arAIN_53.dblValue;

(* [A1-10, AI6-7]  Напряжение питания ШУ, резервный ввод *)
fb_TokStatora(arAIN := arAIN_65, strAI := ai.Tok_statora, err_mod:=arERR_9);
AI_65_dblValue := arAIN_65.dblValue;

A1_10_err_mode := arERR_9.wValue;

(* ---- proc_AI_Init.st ---- *)
FUNCTION_BLOCK proc_AI_Init

VAR_INPUT
	init : BOOL; (*Флаг необходимости инициализации структур-дескрипторов.*)
END_VAR

VAR
	stAI_Ini : fb_AI_Init; (*ФБ инициализации структуры-дескриптора для канала AI.*)
	inits : UINT; (*Текущее количество успешно проинициализированных структур-дескрипторов.*)
END_VAR

VAR_INPUT
	initiales : UINT; (*Общее количество успешно проинициализированных структур-дескрипторов.*)
END_VAR

VAR_EXTERNAL
	ai : AiConfig;
END_VAR

inits := 0; (* Флаг необходимости инициализации структур-дескрипторов *)

(********************************************* Модуль A2-14 ******************************************************)
(* [A2-14, AI0-0] TStalisStatoraKanal1 *)
stAI_Ini(data_Ini := TRUE, dLL := 0.0, dHL := 150.0,
ISVALIDREF_HW := TRUE, dHW := 130.0, aperturFilter:= 0.5,
strAI := ai.Tstali_statora_kanal_1);
inits := inits + BOOL_TO_UINT(stAI_Ini.Init);

(* [A2-14, AI0-1] TStalisStatoraKanal2 *)
stAI_Ini(data_Ini := TRUE,  dLL := 0.0, dHL := 150.0,
ISVALIDREF_HW := TRUE, dHW := 130.0, aperturFilter:= 0.5,
strAI := ai.Tstali_statora_kanal_2);
inits := inits + BOOL_TO_UINT(stAI_Ini.Init);

(* [A2-14, AI0-2] TStalisStatoraKanal3 *)
stAI_Ini(data_Ini := TRUE,  dLL := 0.0, dHL :=150.0,
ISVALIDREF_HW := TRUE, dHW := 130.0, aperturFilter:= 0.5,
strAI := ai.Tstali_statora_kanal_3);
inits := inits + BOOL_TO_UINT(stAI_Ini.Init);

(* [A2-14, AI0-3] TMediStatoraKanal1 *)
stAI_Ini(data_Ini := TRUE,  dLL := 0.0, dHL := 150.0,
ISVALIDREF_HW := TRUE, dHW := 130.0, aperturFilter:= 0.5,
strAI := ai.Tmedi_statora_kanal_1);
inits := inits + BOOL_TO_UINT(stAI_Ini.Init);

(********************************************* Модуль A2-15 ******************************************************)

(* [A2-15, AI1-0] TMediStatoraKanal2 *)
stAI_Ini(data_Ini :=TRUE,  dLL := 0.0, dHL := 150.0,
ISVALIDREF_HW := TRUE, dHW := 130.0, aperturFilter:= 0.5,
strAI := ai.Tmedi_statora_kanal_2);
inits := inits + BOOL_TO_UINT(stAI_Ini.Init);

(* [A2-15, AI1-1] TMediStatoraKanal3 *)
stAI_Ini(data_Ini := TRUE,  dLL := 0.0, dHL := 150.0,
ISVALIDREF_HW := TRUE, dHW := 130.0, aperturFilter:= 0.5,
strAI := ai.Tmedi_statora_kanal_3);
inits := inits + BOOL_TO_UINT(stAI_Ini.Init);

(* [A2-15, AI1-2] TOpornogoPodshipnikaEDT_1 *)
stAI_Ini(data_Ini := TRUE,  dLL := 0.0, dHL := 100.0,
ISVALIDREF_HA := TRUE, ISVALIDREF_HW := TRUE, dHA := 80.0, dHW := 75.0, aperturFilter:= 0.5, dMaxChangeSpeed := 10.0,
strAI := ai.Toporno_podshipnika_EDT_1);
inits := inits + BOOL_TO_UINT(stAI_Ini.Init);

(* [A2-15, AI1-3]  TOpornoYpornogoPodshipnikaEDT_2 *)
stAI_Ini(data_Ini := TRUE,  dLL := 0.0, dHL := 100.0,
ISVALIDREF_HA := TRUE, ISVALIDREF_HW := TRUE, dHA := 80.0, dHW := 75.0, aperturFilter:= 0.5, dMaxChangeSpeed := 10.0,
strAI := ai.Toy_podshipnika_EDT_2);
inits := inits + BOOL_TO_UINT(stAI_Ini.Init);

(********************************************* Модуль A3-1 ******************************************************)

(* [A3-1, AI2-0]  TOpornoYpornogoPodshipnikaKolesaRedEDT_3 *)
stAI_Ini(data_Ini := TRUE,  dLL := 0.0, dHL := 100.0,
ISVALIDREF_HA := TRUE, ISVALIDREF_HW := TRUE, dHA := 80.0, dHW := 75.0, aperturFilter:= 0.5, dMaxChangeSpeed := 10.0,
strAI := ai.Toy_podshipnika_kol_EDT_3);
inits := inits + BOOL_TO_UINT(stAI_Ini.Init);

(* [A3-1, AI2-1] TOpornoYpornogoPodshipnikaKolesaRedHT_4 *)
stAI_Ini(data_Ini := TRUE,  dLL := 0.0, dHL := 100.0,
ISVALIDREF_HA := TRUE, ISVALIDREF_HW := TRUE, dHA := 80.0, dHW := 75.0, aperturFilter:= 0.5, dMaxChangeSpeed := 10.0,
strAI := ai.Toy_podshipnika_kol_EDT_4);
inits := inits + BOOL_TO_UINT(stAI_Ini.Init);

(* [A3-1, AI2-2] TOpornogoPodshipnikaShesterniReduktoraT_5 *)
stAI_Ini(data_Ini := TRUE,  dLL := 0.0, dHL := 100.0,
ISVALIDREF_HA := TRUE, ISVALIDREF_HW := TRUE, dHA := 80.0, dHW := 75.0, aperturFilter:= 0.5, dMaxChangeSpeed := 10.0,
strAI := ai.Toy_podshipnika_shest_red_EDT_5);
inits := inits + BOOL_TO_UINT(stAI_Ini.Init);

(* [A3-1, AI2-3] TOpornogoPodshipnikaReduktoraHT_6 *)
stAI_Ini(data_Ini := TRUE,  dLL := 0.0, dHL := 100.0,
ISVALIDREF_HA := TRUE, ISVALIDREF_HW := TRUE, dHA := 80.0, dHW := 75.0, aperturFilter:= 0.5, dMaxChangeSpeed := 10.0,
strAI := ai.Ty_podshipnika_red_EDT_6);
inits := inits + BOOL_TO_UINT(stAI_Ini.Init);

(********************************************* Модуль A3-2 ******************************************************)

(* [A3-2, AI3-01]  TOpornoYpornogoPodshipnikaNagnetateljaT_7_1 *)
stAI_Ini(data_Ini := TRUE,  dLL := 0.0, dHL := 100.0,
ISVALIDREF_HA := TRUE, ISVALIDREF_HW := TRUE, dHA := 80.0, dHW := 75.0, aperturFilter:= 0.5, dMaxChangeSpeed := 10.0,
strAI := ai.Ty_podshipnika_nagnet_EDT_7_1);
inits := inits + BOOL_TO_UINT(stAI_Ini.Init);

(* [A3-2, AI3-01]  TOpornoYpornogoPodshipnikaNagnetateljaT_7_2 *)
stAI_Ini(data_Ini := TRUE,  dLL := 0.0, dHL := 100.0,
ISVALIDREF_HA := TRUE, ISVALIDREF_HW := TRUE, dHA := 80.0, dHW := 75.0, aperturFilter:= 0.5, dMaxChangeSpeed := 10.0,
strAI := ai.Ty_podshipnika_nagnet_EDT_7_2);
inits := inits + BOOL_TO_UINT(stAI_Ini.Init);

(* [A3-2, AI3-2]  TOpornoYpornogoPodshipnikaSvobodnogoKoncaNT_8_1 *)
stAI_Ini(data_Ini := TRUE,  dLL := 0.0, dHL := 100.0,
ISVALIDREF_HA := TRUE, ISVALIDREF_HW := TRUE, dHA := 80.0, dHW := 75.0, aperturFilter:= 0.5, dMaxChangeSpeed := 10.0,
strAI := ai.Toy_podshipnika_svobod_konca_EDT_8_1);
inits := inits + BOOL_TO_UINT(stAI_Ini.Init);

(* [A3-2, AI3-2]  TOpornoYpornogoPodshipnikaSvobodnogoKoncaNT_8_2 *)
stAI_Ini(data_Ini := TRUE,  dLL := 0.0, dHL := 100.0,
ISVALIDREF_HA := TRUE, ISVALIDREF_HW := TRUE, dHA := 80.0, dHW := 75.0, aperturFilter:= 0.5, dMaxChangeSpeed := 10.0,
strAI := ai.Toy_podshipnika_svobod_konca_EDT_8_2);
inits := inits + BOOL_TO_UINT(stAI_Ini.Init);

(********************************************* Модуль A3-3 ******************************************************)

(* [A3-3, AI4-1]  TYpornogoPodshipnikaRavKolodokHT_9_1 *)
stAI_Ini(data_Ini := TRUE,  dLL := 0.0, dHL := 100.0,
ISVALIDREF_HA := TRUE, ISVALIDREF_HW := TRUE, dHA := 80.0, dHW := 75.0, aperturFilter:= 0.5, dMaxChangeSpeed := 10.0,
strAI := ai.Toy_podshipnika_rab_kol_EDT_9_1);
inits := inits + BOOL_TO_UINT(stAI_Ini.Init);

(* [A3-3, AI4-1]  TYpornogoPodshipnikaRavKolodokHT_9_2 *)
stAI_Ini(data_Ini := TRUE,  dLL := 0.0, dHL := 100.0,
ISVALIDREF_HA := TRUE, ISVALIDREF_HW := TRUE, dHA := 80.0, dHW := 75.0, aperturFilter:= 0.5, dMaxChangeSpeed := 10.0,
strAI := ai.Toy_podshipnika_rab_kol_EDT_9_2);
inits := inits + BOOL_TO_UINT(stAI_Ini.Init);

(* [A3-3, AI4-3] TYpornogoPodshipnikaNerabKolodokHT_10_1 *)
stAI_Ini(data_Ini := TRUE,  dLL := 0.0, dHL := 100.0,
ISVALIDREF_HA := TRUE, ISVALIDREF_HW := TRUE, dHA := 80.0, dHW := 75.0, aperturFilter:= 0.5, dMaxChangeSpeed := 10.0,
strAI := ai.Toy_podshipnika_nerab_kol_EDT_10_1);
inits := inits + BOOL_TO_UINT(stAI_Ini.Init);

(* [A3-3, AI4-3] TYpornogoPodshipnikaNerabKolodokHT_10_2 *)
stAI_Ini(data_Ini := TRUE,  dLL := 0.0, dHL := 100.0,
ISVALIDREF_HA := TRUE, ISVALIDREF_HW := TRUE, dHA := 80.0, dHW := 75.0, aperturFilter:= 0.5, dMaxChangeSpeed := 10.0,
strAI := ai.Toy_podshipnika_nerab_kol_EDT_10_2);
inits := inits + BOOL_TO_UINT(stAI_Ini.Init);

(********************************************* Модуль A3-4 ******************************************************)
(* [A3-4, AI5-0] THolodnogoVozduhaEDKanall *)
stAI_Ini(data_Ini := TRUE,  dLL := 0.0, dHL := 100.0,
ISVALIDREF_HW := TRUE, dHW := 60.0, aperturFilter:= 0.5,
strAI := ai.Tholodnogo_vozduha_ED_kanal_1);
inits := inits + BOOL_TO_UINT(stAI_Ini.Init);

(* [A3-4, AI5-1] THolodnogoVozduhaEDKanal2 *)
stAI_Ini(data_Ini := TRUE,  dLL := 0.0, dHL := 100.0,
ISVALIDREF_HW := TRUE, dHW := 60.0, aperturFilter:= 0.5,
strAI := ai.Tholodnogo_vozduha_ED_kanal_2);
inits := inits + BOOL_TO_UINT(stAI_Ini.Init);

(* [A3-4, AI5-2]  TGorjachegoVozduhaEDKanall *)
stAI_Ini(data_Ini := TRUE,  dLL := 0.0, dHL := 100.0,
ISVALIDREF_HW := TRUE, dHW := 70.0, aperturFilter:= 0.5,
strAI := ai.Tgorjachego_vozduha_ED_kanal_1);
inits := inits + BOOL_TO_UINT(stAI_Ini.Init);

(* [A3-4, AI5-3] TGorjachegoVozduhaEDKanal2 *)
stAI_Ini(data_Ini := TRUE,  dLL := 0.0, dHL := 100.0,
ISVALIDREF_HW := TRUE, dHW := 70.0, aperturFilter:= 0.5,
strAI := ai.Tgorjachego_vozduha_ED_kanal_2);
inits := inits + BOOL_TO_UINT(stAI_Ini.Init);

(********************************************* Модуль A3-5 ******************************************************)

(* [A3-5, AI6-0] TNArujnogoVozduha *)
stAI_Ini(data_Ini := TRUE,  dLL := -50.0, dHL := 100.0,
ISVALIDREF_HW := TRUE, dHW := 70.0, aperturFilter:= 0.5,
strAI := ai.Tnarujnogo_vozduha);
inits := inits + BOOL_TO_UINT(stAI_Ini.Init);

(* [A3-5, AI6-1]  TgazaNaVhodeH *)
stAI_Ini(data_Ini := TRUE,  dLL := -50.0, dHL := 100.0,
ISVALIDREF_HW := TRUE, dHW := 80.0, aperturFilter:= 0.5,
strAI := ai.Tgaza_na_vhode_H);
inits := inits + BOOL_TO_UINT(stAI_Ini.Init);

(* [A3-5, AI6-2] TgazaNaVyhodeH *)
stAI_Ini(data_Ini := TRUE,  dLL := -50.0, dHL := 100.0,
ISVALIDREF_HW := TRUE, ISVALIDREF_HA := TRUE, dHa :=90.0, dHW := 80.0, aperturFilter:= 0.5, dMaxChangeSpeed := 10.0,
strAI := ai.Tgaza_na_vyhode_H);
inits := inits + BOOL_TO_UINT(stAI_Ini.Init);

(********************************************* Модуль A3-6 ******************************************************)
(* [A3-6, AI7-0] TMasladoAVOM *)
stAI_Ini(data_Ini := TRUE,  dLL := 0.0, dHL := 150.0,
ISVALIDREF_HW := TRUE, dHW := 55.0, aperturFilter:= 0.5,
strAI := ai.Tmasla_do_AVOM);
inits := inits + BOOL_TO_UINT(stAI_Ini.Init);

(* [A3-6, AI7-1] TMaslaPosleAVOM *)
stAI_Ini(data_Ini := TRUE,  dLL := 0.0, dHL := 150.0,
ISVALIDREF_HW := TRUE, dHW := 55.0, aperturFilter:= 0.5, dMaxChangeSpeed := 10.0,
strAI := ai.Tmasla_posle_AVOM);
inits := inits + BOOL_TO_UINT(stAI_Ini.Init);
(********************************************* Модуль A3-8 ******************************************************)
(* [A3-8, AI9-0]  TMaslaMB *)
stAI_Ini(data_Ini := TRUE,  dLL := 0.0, dHL := 150.0,
ISVALIDREF_LW := TRUE, dLW := 25.0, aperturFilter:= 0.5, dMaxChangeSpeed := 10.0,
strAI := ai.Tmasla_MB);
inits := inits + BOOL_TO_UINT(stAI_Ini.Init);

(* [A3-6, AI7-2] TMaslaMB_TEN *)
stAI_Ini(data_Ini := TRUE,  dLL := 0.0, dHL := 100.0,
ISVALIDREF_HW := TRUE, dHW := 50.0, aperturFilter:= 0.5, dMaxChangeSpeed := 10.0,
strAI := ai.Tmasla_MB_TEN);
inits := inits + BOOL_TO_UINT(stAI_Ini.Init);

(* [A3-8, AI9-1]  TEmperatura_v_SHU *)
stAI_Ini(data_Ini := TRUE,  dLL := -40.0, dHL := 100.0, CurrentShotCircuit := 20320.0, CurrentBreakCircuit := 3680.0,
aperturFilter:= 0.5, strAI := ai.Tshu);
inits := inits + BOOL_TO_UINT(stAI_Ini.Init);

(* [A3-8, AI9-2]  DavlenijaMasloSmNizkoe *)
stAI_Ini(data_Ini := TRUE,  dLL := 0.0, dHL := 250.0,
ISVALIDREF_LW := TRUE, ISVALIDREF_LA := TRUE, dLW := 50.0, dLA := 25.0,  CurrentShotCircuit := 20240.0, CurrentBreakCircuit := 3760.0,  aperturFilter:= 0.5,
strAI := ai.Pmaslo_sm_nizkoe);
inits := inits + BOOL_TO_UINT(stAI_Ini.Init);

(* [A3-8, AI9-3]  PerepadDavlenieNaMasloFiltre *)
stAI_Ini(data_Ini := TRUE,  dLL := 0.0, dHL := 250.0,
ISVALIDREF_HW := TRUE, dHW := 150.0, CurrentShotCircuit := 20240.0, CurrentBreakCircuit := 3760.0, aperturFilter:= 0.5,
strAI := ai.dPgaza_na_maslo_filtre);
inits := inits + BOOL_TO_UINT(stAI_Ini.Init);

(********************************************* Модуль A3-9 ******************************************************)
(* [A3-9, AI10-0]  DavlenijaMasloSmVysokoe *)
stAI_Ini(data_Ini := TRUE,  dLL := 0.0, dHL := 1000.0,
ISVALIDREF_LW := TRUE, ISVALIDREF_LA := TRUE, dLW := 300.0, dLA := 250.0, CurrentShotCircuit := 20240.0, CurrentBreakCircuit := 3760.0, aperturFilter:= 0.5,
strAI := ai.Pmaslo_sm_vysokoe);
inits := inits + BOOL_TO_UINT(stAI_Ini.Init);

(* [A3-9, AI10-1]  DavlenijaMaslaPosleGNS *)
stAI_Ini(data_Ini := TRUE,  dLL := 0.0, dHL := 250.0, aperturFilter:= 0.5, CurrentShotCircuit := 20240.0, CurrentBreakCircuit := 3760.0,
ISVALIDREF_LW := TRUE, ISVALIDREF_HW := TRUE,
dLW := 187.0, dHW := 242.0,
strAI := ai.Pmasla_posle_GNS);
inits := inits + BOOL_TO_UINT(stAI_Ini.Init);

(* [A3-9, AI10-2] DavlenijaMaslaPosleNU *)
stAI_Ini(data_Ini := TRUE,  dLL := 0.0, dHL := 10.0, aperturFilter:= 0.5, CurrentShotCircuit := 20240.0, CurrentBreakCircuit := 3760.0,
ISVALIDREF_LW := TRUE, dLW := 3.0,
strAI := ai.Pmasla_posle_NU);
inits := inits + BOOL_TO_UINT(stAI_Ini.Init);

(********************************************* Модуль A3-10 ******************************************************)
(* [A3-10, AI11-0] PerepadDavlenieNaKonfuzore *)
stAI_Ini(data_Ini := TRUE,  dLL := 0.0, dHL := 250.0,
ISVALIDREF_LW := TRUE, dLW := 15.0, aperturFilter:= 0.5, CurrentShotCircuit := 20240.0, CurrentBreakCircuit := 3760.0,
strAI := ai.dPgaza_na_konfuzore);
inits := inits + BOOL_TO_UINT(stAI_Ini.Init);

(* [A3-10, AI11-1] OsSdvigNagnetatelja_Plus *)
stAI_Ini(data_Ini := TRUE,  dLL := 0.0, dHL := 1000.0,
ISVALIDREF_HA := TRUE, ISVALIDREF_HW := TRUE, dHW := 200.0, dHA := 300.0, aperturFilter := 0.5, CurrentShotCircuit := 20240.0, CurrentBreakCircuit := 3760.0,
strAI := ai.Os_sdvig_nagnetatelja_plus);
inits := inits + BOOL_TO_UINT(stAI_Ini.Init);

(* [A3-10, AI11-2] OsSdvigNagnetatelja_Minus *)
stAI_Ini(data_Ini := TRUE,  dLL := 0.0, dHL := 1600.0,
ISVALIDREF_LW := TRUE, dLW := 150.0, ISVALIDREF_LA := TRUE, dLA := 100.0, aperturFilter := 0.5, CurrentShotCircuit := 20240.0, CurrentBreakCircuit := 3760.0,
strAI := ai.Os_sdvig_nagnetatelja_minus);
inits := inits + BOOL_TO_UINT(stAI_Ini.Init);

(* [A3-10, AI11-3] PerepadDavlenieMasloGaz *)
stAI_Ini(data_Ini := TRUE, dLL := 0.0, dHL := 1600.0,
ISVALIDREF_LW := TRUE, ISVALIDREF_LA := TRUE, dLW := 150.0, dLa := 100.0, aperturFilter:= 0.5, CurrentShotCircuit := 20240.0, CurrentBreakCircuit := 3760.0,
strAI := ai.dPmaslo_gaz);
inits := inits + BOOL_TO_UINT(stAI_Ini.Init);

(********************************************* Модуль A3-11 ******************************************************)
(* [A3-11, AI12-0]  DGazaNaVhodeNagnetatelja *)
stAI_Ini(data_Ini := TRUE,  dLL := 0.0, dHL := 10.0,
ISVALIDREF_LW := TRUE, dLW := 4.895, aperturFilter := 0.5, CurrentShotCircuit := 20240.0, CurrentBreakCircuit := 3760.0,
strAI := ai.Pgaza_na_vhode_nagnetatelia);
inits := inits + BOOL_TO_UINT(stAI_Ini.Init);

(* [A3-11, AI12-1]  DGazaNaVyhodeNagnetatelja *)
stAI_Ini(data_Ini := TRUE,  dLL := 0.0, dHL := 10.0,
ISVALIDREF_HA := TRUE, ISVALIDREF_HW := TRUE, dLA := 7.653, dHW := 7.55, aperturFilter := 0.5, CurrentShotCircuit := 20240.0, CurrentBreakCircuit := 3760.0,
strAI := ai.Pgaza_na_vyhode_nagnetatelia);
inits := inits + BOOL_TO_UINT(stAI_Ini.Init);

(* [A3-11, AI12-3]  DavlenieImpulsGaz *)
stAI_Ini(data_Ini := TRUE,  dLL := 0.0, dHL := 10.0,
ISVALIDREF_LW := TRUE, dLW := 5.0, aperturFilter := 0.5, CurrentShotCircuit := 20240.0, CurrentBreakCircuit := 3760.0,
strAI := ai.Pimpuls_gaz);
inits := inits + BOOL_TO_UINT(stAI_Ini.Init);

(********************************************* Модуль A3-12 ******************************************************)
(* [A3-12, AI13-0] YrovenMaslaMB *)
stAI_Ini(data_Ini := TRUE,  dLL := 190.0, dHL := 885.0,
ISVALIDREF_LW := TRUE, dLW := 530.0, aperturFilter := 0.5,  CurrentShotCircuit := 20240.0, CurrentBreakCircuit := 3760.0,
strAI := ai.Yroven_masla_MB);
inits := inits + BOOL_TO_UINT(stAI_Ini.Init);

(********************************************* Модуль A3-13 ******************************************************)
(* [A3-13, AI14-0]  Kontrol_per220V *)
stAI_Ini(data_Ini := TRUE,  dLL := 0.0, dHL := 250.0,
ISVALIDREF_LW := TRUE, ISVALIDREF_HW := TRUE, dLW := 187.0, dHW := 242.0, aperturFilter := 0.5, CurrentShotCircuit := 20240.0, CurrentBreakCircuit := 3760.0,
strAI := ai.Kontrol_per_220V);
inits := inits + BOOL_TO_UINT(stAI_Ini.Init);

(* [A3-13, AI14-1]  Kontrol_post220V *)
stAI_Ini(data_Ini := TRUE,  dLL := 0.0, dHL := 250.0,
ISVALIDREF_HW := TRUE, ISVALIDREF_LW := TRUE, dHW := 242.0, dLW := 187.0, aperturFilter := 0.5, CurrentShotCircuit := 20240.0, CurrentBreakCircuit := 3760.0,
strAI := ai.Kontrol_post_220V);
inits := inits + BOOL_TO_UINT(stAI_Ini.Init);

(* [A3-13, AI14-2]  VibroSkorostOPED_T1 *)
stAI_Ini(data_Ini := TRUE,  dLL := 0.0, dHL := 25.0,
ISVALIDREF_HW := TRUE, ISVALIDREF_HA := TRUE, dHW := 11.0, dHA := 18.0, aperturFilter := 0.5, CurrentShotCircuit := 20240.0, CurrentBreakCircuit := 3760.0,
strAI := ai.Vibro_skorost_OPED_T1);
inits := inits + BOOL_TO_UINT(stAI_Ini.Init);

(* [A3-13, AI14-3]  VibroSkorostOYPED_T2 *)
stAI_Ini(data_Ini := TRUE,  dLL := 0.0, dHL := 25.0,
ISVALIDREF_HW := TRUE, ISVALIDREF_HA := TRUE, dHW := 11.0, dHA := 18.0, aperturFilter := 0.5, CurrentShotCircuit := 20240.0, CurrentBreakCircuit := 3760.0,
strAI := ai.Vibro_skorost_OYPED_T2);
inits := inits + BOOL_TO_UINT(stAI_Ini.Init);

(********************************************* Модуль A3-14 ******************************************************)
(* [A3-14, AI15-0]  VibroSkorostOYPKolesaED_T3 *)
stAI_Ini(data_Ini := TRUE,  dLL := 0.0, dHL := 25.0,
ISVALIDREF_HW := TRUE, ISVALIDREF_HA := TRUE, dHW := 11.0, dHA := 18.0, aperturFilter := 0.5, CurrentShotCircuit := 20240.0, CurrentBreakCircuit := 3760.0,
strAI := ai.Vibro_skorost_OYP_kolesa_ED_T3);
inits := inits + BOOL_TO_UINT(stAI_Ini.Init);

(* [A3-14, AI15-1]  VibroSkorostOPKolesaRH_T4 *)
stAI_Ini(data_Ini := TRUE,  dLL := 0.0, dHL := 25.0,
ISVALIDREF_HW := TRUE, ISVALIDREF_HA := TRUE, dHW := 11.0, dHA := 18.0, aperturFilter := 0.5, CurrentShotCircuit := 20240.0, CurrentBreakCircuit := 3760.0,
strAI := ai.Vibro_skorost_OP_kolesa_RH_T4);
inits := inits + BOOL_TO_UINT(stAI_Ini.Init);

(* [A3-11, AI12-2]  VibroSkorostOPShesterniRED_T5 *)
stAI_Ini(data_Ini := TRUE,  dLL := 0.0, dHL := 25.0,
ISVALIDREF_HW := TRUE, ISVALIDREF_HA := TRUE, dHW := 11.0, dHA := 18.0, aperturFilter := 0.5, CurrentShotCircuit := 20240.0, CurrentBreakCircuit := 3760.0,
strAI := ai.Vibro_skorost_OP_shesterni_RED_T5);
inits := inits + BOOL_TO_UINT(stAI_Ini.Init);

(* [A3-11, AI12-2]  VibroSkorostOPShesterniRED_T5 *)
stAI_Ini(data_Ini := TRUE,  dLL := 0.0, dHL := 25.0,
ISVALIDREF_HW := TRUE, ISVALIDREF_HA := TRUE, dHW := 11.0, dHA := 18.0, aperturFilter := 0.5, CurrentShotCircuit := 20240.0, CurrentBreakCircuit := 3760.0,
strAI := ai.Vibro_skorost_OP_shesterni_RED_T6);
inits := inits + BOOL_TO_UINT(stAI_Ini.Init);

(* [A3-11, AI12-2]  VibroSkorostOPShesterniRED_T5 *)
stAI_Ini(data_Ini := TRUE,  dLL := 0.0, dHL := 1000.0,
ISVALIDREF_LW := TRUE, dLW := 300.0, aperturFilter := 0.5, CurrentShotCircuit := 20240.0, CurrentBreakCircuit := 3760.0,
strAI := ai.Tok_statora);
inits := inits + BOOL_TO_UINT(stAI_Ini.Init);

initiales := 0;
IF init THEN initiales := inits; END_IF;

(* ---- proc_algoritms.st ---- *)
FUNCTION_BLOCK proc_algoritms

VAR
	fb_RemontAlg : RemontAlg;
	fb_TestProtectionAlg : TestProtectionAlg;
	fb_TestImAlg : TestImAlg;
	fb_AutoTen : fb_AutoTenAlg;
	fb_AutoPns : fb_AutoPnsAlg;
	fb_AutoAvom : fb_AutoAvomAlg;
	fb_vibegPNS : fb_vibegPNSAlg;
	fb_AutoNU : fb_AutoNUAlg;
	fb_puskOilSystem : fb_puskOilSystemAlg;
	fb_AntiPompag : fb_AntiPompagAlg;
	fb_NOAlg : NOAlg;
	fb_AOAlg : AOAlg;
	fb_ppuALG : ppuAlg;
	fb_fillingAlg : fillingAlg;
	fb_engineRunAlg : engineRunAlg;
	fb_puskKalg : puskKalg;
	fb_puskValg : puskValg;
	fb_testdPmgAlg : testdPmgAlg;
	fb_testPmsAlg : testPmsAlg;
	fb_ApuskAlg : ApuskAlg;
	fb_SemiAutoPuskAlg : SemiAutoPuskAlg;
	fb_Pusk_first_faza1 : Pusk_first_faza1;
	fb_Pusk_first_faza2 : Pusk_first_faza2;
	fb_Pusk_third_faza : Pusk_third_faza;
	fb_Pusk_Prov_PMS : Prov_PMS;
	fb_Prov_opressovka : Prov_opressovka;
	fb_Pusk_second_faza_chastotny : Pusk_second_faza_chastotny;
	fb_Pusk_second_faza_reactor : Pusk_second_faza_reactor;
END_VAR

VAR_EXTERNAL
	algoritms : AlgoritmsConfig;
	AlgQuestions : AlgoritmsQuestions;
	ai : AiConfig;
	IM : ImConfig;
	AlgTimers : struct_AlgTimers;
END_VAR

fb_RemontAlg(StrAlg:=algoritms.Remont);

fb_TestProtectionAlg(StrAlg:=algoritms.TestProtection);

fb_TestImAlg(StrAlg:=algoritms.testIm);

(*fb_AutoTen(StrAlg:= algoritms.AutoTen,
T_masla:= ai.Toporno_podshipnika_EDT_1,
Uroven_masla:= ai.Yroven_masla_MB,
offTemperature:= Im.AutoTen_offTemperature,
TEN:= Im.Ten,
PNS:= Im.pns);*)

(*fb_AutoPns(StrAlg:= algoritms.AutoPns,
Poil:= ai.Pmasla_posle_GNS,
Ust_Run:= Im.AutoPns_UstRun,
Ust_Stop:= Im.AutoPns_UstStop,
Nasos:= Im.pns,
diPlow:= Im.SingleSignals.P_oil_low);*)

(*fb_AutoAvom(StrAlg:= algoritms.AutoAvom,
im1:= Im.v1_Avom,
im2:= Im.v2_Avom,
on1Temperature:= Im.AutoAvom_onTemp1,
on2Temperature:= Im.AutoAvom_onTemp2,
hystereses:= Im.AutoAvom_hysteresis,
ai:= ai.Tnarujnogo_vozduha);*)

fb_vibegPNS(StrAlg:=algoritms.vibegPNS,
algContinue:=AlgQuestions.vibegPNS_algContinue
);

(*fb_AutoNU(StrAlg:=algoritms.autoNu,
nu1:=Im.nu1,
nu2:=Im.nu2,
Ust_Swap:= Im.AutoNU_Ust_Swap,
mainNU:= Im.AutoNU_mainNU,
dPoil:=ai.Tmasla_MB,
Lowdp_di:=Im.SingleSignals.dP_oilgaz_low
);*)

fb_puskOilSystem(StrAlg:=algoritms.puskOilSystem);

(*fb_AntiPompag(StrAlg:=algoritms.AntiPompag,
Rashod:= ai.Vibro_skorost_OP_shesterni_RED_T6,
Zapas:= ai.Vibro_skorost_OP_shesterni_RED_T5,
P_gasIn:=ai.dPgaza_na_maslo_filtre,
T_gasIn:=ai.Tgaza_na_vhode_H,
dP_konf:=ai.dPgaza_na_konfuzore,
Kran6:= im.Kran6,
UgolVNA:= im.AntiPompag_UgolVNA,
K:=im.AntiPompag_K,
A:=im.AntiPompag_A,
y0:=im.AntiPompag_y0);*)

fb_NOAlg(StrAlg:=algoritms.no);

fb_AOAlg(StrAlg:=algoritms.ao);

fb_ppuAlg(StrAlg:=algoritms.ppu);

fb_fillingAlg(StrAlg:=algoritms.filling);

fb_engineRunAlg(StrAlg:=algoritms.engineRun);

fb_puskKalg(StrAlg:=algoritms.puskK,
questionFilling:=AlgQuestions.puskK_questionFilling,
 questionUnload:=AlgQuestions.puskK_questionUnload
);

fb_puskValg(StrAlg:=algoritms.puskV,
 questionEngine:=AlgQuestions.puskV_questionEngine,
  questionMVoff:=AlgQuestions.puskV_questionMVoff
);

fb_testdPmgAlg(StrAlg:=algoritms.testdPmg,
 algContinue:=AlgQuestions.testdPmg_algContinue
);

fb_testPmsAlg(StrAlg:=algoritms.testPms,
 algContinue:=AlgQuestions.testPms_algContinue
);

fb_ApuskAlg(StrAlg:=algoritms.Apusk);

fb_SemiAutoPuskAlg(StrAlg:=algoritms.SemiAutoPusk,
 cmdRun1ph:=AlgQuestions.SemiAutoPusk_cmdRun1ph,
 cmdRun2ph:=AlgQuestions.SemiAutoPusk_cmdRun2ph,
 cmdRun3ph:=AlgQuestions.SemiAutoPusk_cmdRun3ph
);

fb_Pusk_first_faza1(Stralg:=algoritms.Pusk_F_faza1);

fb_Pusk_first_faza2(Stralg:=algoritms.Pusk_F_faza2);

fb_Pusk_third_faza(Stralg:=algoritms.Pusk_TH_faza);

fb_Pusk_Prov_PMS(Stralg:=algoritms.Prov_PMS_ALG);

fb_Prov_opressovka(Stralg:=algoritms.Prov_opressovka_ALG);

fb_Pusk_second_faza_chastotny(Stralg:=algoritms.Pusk_SEC_faza_chastotny);

fb_Pusk_second_faza_reactor(Stralg:=algoritms.Pusk_SEC_faza_reactor);

(* ---- proc_AO.st ---- *)
FUNCTION_BLOCK proc_AO

VAR
	fb_Reserv_AO_1 : fb_AOSourceMlp; (*[A1-14:1, AI0] Резерв*)
	fb_Reserv_AO_2 : fb_AOSourceMlp; (*[A1-14:2, AI1] Резерв*)
END_VAR

VAR_EXTERNAL
	ao : AOConfig;
	arAOUT_0 : TDoubleData;
	arAOUT_1 : TDoubleData;
END_VAR

(* Циклический опрос. Входные аналоговые параметры *)

(* Модуль A10 *)

(* [A10-1, AO0] Резерв (A10) *)
fb_Reserv_AO_1(OutCurrent := arAOUT_0, strAO := ao.Reserv_AO_1);

(* [A10-1, AO1] Резерв (A10) *)
fb_Reserv_AO_2(OutCurrent := arAOUT_1, strAO := ao.Reserv_AO_2);

(* ---- proc_AO_Init.st ---- *)
FUNCTION_BLOCK proc_AO_Init

VAR_INPUT
	init : BOOL; (*Флаг необходимости инициализации структур-дескрипторов.*)
END_VAR

VAR
	stAO_Ini : fb_AO_Init; (*ФБ инициализации структуры-дескриптора для канала AI.*)
	inits : UINT; (*Текущее количество успешно проинициализированных структур-дескрипторов.*)
END_VAR

VAR_INPUT
	initiales : UINT; (*Общее количество успешно проинициализированных структур-дескрипторов.*)
END_VAR

VAR_EXTERNAL
	ao : AOConfig;
END_VAR

(* Инициализация начало. Входные аналоговые параметры *)

inits := 0; (* Флаг необходимости инициализации структур-дескрипторов *)

(* Модуль A10 *)
(* [A10, AO0] Резерв (A) *)
stAO_Ini(data_Ini := TRUE, (*outLL := 4000.0, outHL := 20000.0,*)
  newLL_ISVALIDREF := TRUE, newHL_ISVALIDREF := TRUE,
  newLL := 0.0, newHL := 100.0,
  strAO := ao.Reserv_AO_1);
inits := inits + BOOL_TO_UINT(stAO_Ini.Init);

(* [A1-10, AO1] Резерв (A) *)
stAO_Ini(data_Ini := TRUE, (*outLL := 4000.0, outHL := 20000.0,*)
  (*newLL_ISVALIDREF := TRUE, newHL_ISVALIDREF := TRUE,*)
  (*newLL := 0.0, newHL := 100.0,*)
strAO := ao.Reserv_AO_2);
inits := inits + BOOL_TO_UINT(stAO_Ini.Init);

initiales := 0;
IF init THEN initiales := inits; END_IF;

(* ---- proc_DI.st ---- *)
FUNCTION_BLOCK proc_DI

VAR
	di_0 : fb_DiSourceMlp;
	di_1 : fb_DiSourceMlp;
	di_2 : fb_DiSourceMlp;
	di_3 : fb_DiSourceMlp;
	di_4 : fb_DiSourceMlp;
	di_5 : fb_DiSourceMlp;
	di_6 : fb_DiSourceMlp;
	di_7 : fb_DiSourceMlp;
	di_8 : fb_DiSourceMlp;
	di_9 : fb_DiSourceMlp;
	di_10 : fb_DiSourceMlp;
	di_11 : fb_DiSourceMlp;
	di_12 : fb_DiSourceMlp;
	di_13 : fb_DiSourceMlp;
	di_14 : fb_DiSourceMlp;
	di_15 : fb_DiSourceMlp;
	di_16 : fb_DiSourceMlp;
	di_17 : fb_DiSourceMlp;
	di_18 : fb_DiSourceMlp;
	di_19 : fb_DiSourceMlp;
	di_20 : fb_DiSourceMlp;
	di_21 : fb_DiSourceMlp;
END_VAR

VAR_EXTERNAL
	arDIN_0 : TItemDIN;
	arDIN_1 : TItemDIN;
	arDIN_2 : TItemDIN;
	arDIN_3 : TItemDIN;
	arDIN_4 : TItemDIN;
	arDIN_5 : TItemDIN;
	arDIN_6 : TItemDIN;
	arDIN_7 : TItemDIN;
	arDIN_8 : TItemDIN;
	arDIN_9 : TItemDIN;
	arDIN_10 : TItemDIN;
	arDIN_11 : TItemDIN;
	arDIN_12 : TItemDIN;
	arDIN_13 : TItemDIN;
	arDIN_14 : TItemDIN;
	arDIN_15 : TItemDIN;
	arDIN_16 : TItemDIN;
	arDIN_17 : TItemDIN;
	arDIN_18 : TItemDIN;
	arDIN_19 : TItemDIN;
	arDIN_20 : TItemDIN;
	arDIN_21 : TItemDIN;
	di : DiConfig;
	DI_0_1_wValue : UDINT;
	DI_10_11_wValue : UDINT;
	DI_12_13_wValue : UDINT;
	DI_14_15_wValue : UDINT;
	DI_16_17_wValue : UDINT;
	DI_18_19_wValue : UDINT;
	DI_20_21_wValue : UDINT;
	DI_2_3_wValue : UDINT;
	DI_4_5_wValue : UDINT;
	DI_6_7_wValue : UDINT;
	DI_8_9_wValue : UDINT;
	A1_12_err_mode : UINT;
	A1_13_err_mode : UINT;
	A1_14_err_mode : UINT;
	A1_15_err_mode : UINT;
	A2_10_err_mode : UINT;
	A2_4_err_mode : UINT;
	A2_5_err_mode : UINT;
	A2_6_err_mode : UINT;
	A2_7_err_mode : UINT;
	A2_8_err_mode : UINT;
	A2_9_err_mode : UINT;
	arERR_11 : TItemDIN;
	arERR_12 : TItemDIN;
	arERR_13 : TItemDIN;
	arERR_14 : TItemDIN;
	arERR_18 : TItemDIN;
	arERR_19 : TItemDIN;
	arERR_20 : TItemDIN;
	arERR_21 : TItemDIN;
	arERR_22 : TItemDIN;
	arERR_23 : TItemDIN;
	arERR_24 : TItemDIN;
END_VAR

(* Циклический опрос. Входные дискретные параметры *)
(* Модуль A1-12 *)
di_0(arDIN := arDIN_0, strDI:=di.di_0, err_mod:=arERR_11);
di_1(arDIN := arDIN_1, strDI:=di.di_1, err_mod:=arERR_11);
DI_0_1_wValue:=TwoUint_To_UDINT(arDIN_0.wValue, arDIN_1.wValue);
A1_12_err_mode:= arERR_11.wValue;

(* Модуль A1-13 *)
di_2(arDIN := arDIN_2, strDI:=di.di_2,  err_mod:=arERR_12);
di_3(arDIN := arDIN_3, strDI:=di.di_3,  err_mod:=arERR_12);
DI_2_3_wValue:=TwoUint_To_UDINT(arDIN_2.wValue, arDIN_3.wValue);
A1_13_err_mode:= arERR_12.wValue;

(* Модуль A1-14 *)
di_4(arDIN := arDIN_4, strDI:=di.di_4,  err_mod:=arERR_13);
di_5(arDIN := arDIN_5, strDI:=di.di_5,  err_mod:=arERR_13);
DI_4_5_wValue:=TwoUint_To_UDINT(arDIN_4.wValue, arDIN_5.wValue);
A1_14_err_mode:= arERR_13.wValue;

(* Модуль A1-15 *)
di_6(arDIN := arDIN_6, strDI:=di.di_6,  err_mod:=arERR_14);
di_7(arDIN := arDIN_7, strDI:=di.di_7,  err_mod:=arERR_14);
DI_6_7_wValue:=TwoUint_To_UDINT(arDIN_6.wValue, arDIN_7.wValue);
A1_15_err_mode:= arERR_14.wValue;

(* Модуль A2-4 *)
di_8(arDIN := arDIN_8, strDI:=di.di_8,  err_mod:=arERR_18);
di_9(arDIN := arDIN_9, strDI:=di.di_9,  err_mod:=arERR_18);
DI_8_9_wValue:=TwoUint_To_UDINT(arDIN_8.wValue, arDIN_9.wValue);
A2_4_err_mode:= arERR_18.wValue;

(* Модуль A2-5 *)
di_10(arDIN := arDIN_10, strDI:=di.di_10,  err_mod:=arERR_19);
di_11(arDIN := arDIN_11, strDI:=di.di_11,  err_mod:=arERR_19);
DI_10_11_wValue:=TwoUint_To_UDINT(arDIN_10.wValue, arDIN_11.wValue);
A2_5_err_mode:= arERR_19.wValue;

(* Модуль A2-6 *)
di_12(arDIN := arDIN_12, strDI:=di.di_12,  err_mod:=arERR_20);
di_13(arDIN := arDIN_13, strDI:=di.di_13,  err_mod:=arERR_20);
DI_12_13_wValue:=TwoUint_To_UDINT(arDIN_12.wValue, arDIN_13.wValue);
A2_6_err_mode:= arERR_20.wValue;

(* Модуль A2-7 *)
di_14(arDIN := arDIN_14, strDI:=di.di_14,  err_mod:=arERR_21);
di_15(arDIN := arDIN_15, strDI:=di.di_15,  err_mod:=arERR_21);
DI_14_15_wValue:=TwoUint_To_UDINT(arDIN_14.wValue, arDIN_15.wValue);
A2_7_err_mode:= arERR_21.wValue;

di_16(arDIN := arDIN_16, strDI:=di.di_16,  err_mod:=arERR_22);
di_17(arDIN := arDIN_17, strDI:=di.di_17,  err_mod:=arERR_22);
DI_16_17_wValue:=TwoUint_To_UDINT(arDIN_16.wValue, arDIN_17.wValue);
A2_8_err_mode:= arERR_22.wValue;

di_18(arDIN := arDIN_18, strDI:=di.di_18,  err_mod:=arERR_23);
di_19(arDIN := arDIN_19, strDI:=di.di_19,  err_mod:=arERR_23);
DI_18_19_wValue:=TwoUint_To_UDINT(arDIN_18.wValue, arDIN_19.wValue);
A2_9_err_mode:= arERR_23.wValue;

di_20(arDIN := arDIN_20, strDI:=di.di_20,  err_mod:=arERR_24);
di_21(arDIN := arDIN_21, strDI:=di.di_21,  err_mod:=arERR_24);
DI_20_21_wValue:=TwoUint_To_UDINT(arDIN_20.wValue, arDIN_21.wValue);
A2_10_err_mode:= arERR_24.wValue;

(* ---- proc_DI_Init.st ---- *)
FUNCTION_BLOCK proc_DI_Init

VAR_INPUT
	init : BOOL; (*Флаг необходимости инициализации структур-дескрипторов.*)
END_VAR

VAR
	stDI_Ini : fb_DI_Init; (*ФБ инициализации структуры-дескриптора канала DI.*)
	inits : UINT; (*Текущее количество успешно проинициализированных структур-дескрипторов.*)
END_VAR

VAR_INPUT
	initiales : UINT; (*Общее количество успешно проинициализированных структур-дескрипторов.*)
END_VAR

VAR_EXTERNAL
	di : DiConfig; (*Входные дискретные сигналы*)
END_VAR

(* Инициализация начало. Входные дискретные параметры *)

inits := 0; (* Флаг необходимости инициализации структур-дескрипторов *)

(* Модуль A1-1 *)

stDI_Ini(data_Ini := true, imit:=FALSE, strDI := di.di_0);
inits := inits + BOOL_TO_UINT(stDI_Ini.Init);

stDI_Ini(data_Ini := true, imit:=FALSE, strDI := di.di_1);
inits := inits + BOOL_TO_UINT(stDI_Ini.Init);

(* Модуль A1-2 *)
stDI_Ini(data_Ini := true, imit:=FALSE, strDI := di.di_2);
inits := inits + BOOL_TO_UINT(stDI_Ini.Init);

stDI_Ini(data_Ini := true, imit:=FALSE, strDI := di.di_3);
inits := inits + BOOL_TO_UINT(stDI_Ini.Init);

(* Модуль A1-3 *)
stDI_Ini(data_Ini := true, imit:=FALSE, strDI := di.di_4);
inits := inits + BOOL_TO_UINT(stDI_Ini.Init);

stDI_Ini(data_Ini := true, imit:=FALSE, strDI := di.di_5);
inits := inits + BOOL_TO_UINT(stDI_Ini.Init);

(* Модуль A1-4 *)
stDI_Ini(data_Ini := true, imit:=FALSE, strDI := di.di_6);
inits := inits + BOOL_TO_UINT(stDI_Ini.Init);

stDI_Ini(data_Ini := true, imit:=FALSE, strDI := di.di_7);
inits := inits + BOOL_TO_UINT(stDI_Ini.Init);

(* Модуль A1-5 *)
stDI_Ini(data_Ini := true, imit:=FALSE,  strDI := di.di_8);
inits := inits + BOOL_TO_UINT(stDI_Ini.Init);

stDI_Ini(data_Ini := true, imit:=FALSE,  strDI := di.di_9);
inits := inits + BOOL_TO_UINT(stDI_Ini.Init);

(* Модуль A1-6 *)
stDI_Ini(data_Ini := true, imit:=FALSE,  strDI := di.di_10);
inits := inits + BOOL_TO_UINT(stDI_Ini.Init);

stDI_Ini(data_Ini := true, imit:=FALSE,  strDI := di.di_11);
inits := inits + BOOL_TO_UINT(stDI_Ini.Init);

(* Модуль A1-7 *)
stDI_Ini(data_Ini := true, imit:=FALSE, strDI := di.di_12);
inits := inits + BOOL_TO_UINT(stDI_Ini.Init);

stDI_Ini(data_Ini := true, imit:=FALSE, strDI := di.di_13);
inits := inits + BOOL_TO_UINT(stDI_Ini.Init);

(* Модуль A1-8 *)
stDI_Ini(data_Ini := true, imit:=FALSE, strDI := di.di_14);
inits := inits + BOOL_TO_UINT(stDI_Ini.Init);

stDI_Ini(data_Ini := true, imit:=FALSE, strDI := di.di_16);
inits := inits + BOOL_TO_UINT(stDI_Ini.Init);

stDI_Ini(data_Ini := true, imit:=FALSE, strDI := di.di_17);
inits := inits + BOOL_TO_UINT(stDI_Ini.Init);

stDI_Ini(data_Ini := true, imit:=FALSE, strDI := di.di_18);
inits := inits + BOOL_TO_UINT(stDI_Ini.Init);

stDI_Ini(data_Ini := true, imit:=FALSE, strDI := di.di_19);
inits := inits + BOOL_TO_UINT(stDI_Ini.Init);

stDI_Ini(data_Ini := true, imit:=FALSE, strDI := di.di_20);
inits := inits + BOOL_TO_UINT(stDI_Ini.Init);

stDI_Ini(data_Ini := true, imit:=FALSE, strDI := di.di_21);
inits := inits + BOOL_TO_UINT(stDI_Ini.Init);

initiales := 0;
IF init THEN initiales := inits; END_IF;

(* ---- proc_DO.st ---- *)
FUNCTION_BLOCK proc_DO

VAR
	do_0 : fb_DOSourceMlp;
	do_1 : fb_DOSourceMlp;
	do_2 : fb_DOSourceMlp;
	do_3 : fb_DOSourceMlp;
	do_4 : fb_DOSourceMlp;
	gpio_out : fb_DOSourceMlp;
END_VAR

VAR_EXTERNAL
	od : DOconfig;
	arDOUT_0 : TWordData;
	arDOUT_1 : TWordData;
	arDOUT_2 : TWordData;
	arDOUT_3 : TWordData;
	arDOUT_4 : TWordData;
	arERR_66 : TItemDIN;
	arDOUT_66 : TWordData;
	arERR_0 : TItemDIN;
	arERR_1 : TItemDIN;
	arERR_2 : TItemDIN;
	arERR_15 : TItemDIN;
	arERR_16 : TItemDIN;
	A1_1_err_mode : UINT;
	A1_2_err_mode : UINT;
	A1_3_err_mode : UINT;
	A2_1_err_mode : UINT;
	A2_4_err_mode : UINT;
	DO_0_wValue : UINT;
	DO_1_wValue : UINT;
	DO_2_wValue : UINT;
	DO_3_wValue : UINT;
	DO_4_wValue : UINT;
END_VAR

(* Циклический опрос. Входные дискретные параметры *)

(* Модуль A1-1 *)
do_0(arDout := arDOUT_0, strDO := od.do_0, err_mod:=arERR_0);
DO_0_wValue:=arDOUT_0.wValue;
A1_1_err_mode:= arERR_0.wValue;

(* Модуль A1-2 *)
do_1(arDout := arDOUT_1, strDO := od.do_1, err_mod:=arERR_1);
DO_1_wValue:=arDOUT_1.wValue;
A1_2_err_mode:= arERR_1.wValue;

(* Модуль A1-3 *)
do_2(arDout := arDOUT_2, strDO := od.do_2, err_mod:=arERR_2);
DO_2_wValue:=arDOUT_2.wValue;
A1_3_err_mode:= arERR_2.wValue;

(* Модуль A2-1 *)
do_3(arDout := arDOUT_3, strDO := od.do_3, err_mod:=arERR_15);
DO_3_wValue:=arDOUT_3.wValue;
A2_1_err_mode:= arERR_15.wValue;

(* Модуль A2-1 *)
do_4(arDout := arDOUT_4, strDO := od.do_4, err_mod:=arERR_15);
DO_4_wValue:=arDOUT_4.wValue;
A2_4_err_mode:= arERR_16.wValue;

gpio_out(arDout := arDOUT_66, strDO := od.gpio_out, err_mod:=arERR_66);

(* ---- proc_DO_Init.st ---- *)
FUNCTION_BLOCK proc_DO_Init

VAR_INPUT
	init : BOOL; (*Флаг необходимости инициализации структур-дескрипторов.*)
END_VAR

VAR
	stDO_Ini : fb_DO_Init; (*ФБ инициализации структуры-дескриптора канала DO.*)
	inits : UINT; (*Текущее количество успешно проинициализированных структур-дескрипторов.*)
END_VAR

VAR_INPUT
	initiales : UINT; (*Общее количество успешно проинициализированных структур-дескрипторов.*)
END_VAR

VAR_EXTERNAL
	od : DOconfig; (*Выходные дискретные сигналы*)
END_VAR

(* Инициализация начало. Входные дискретные параметры *)

inits := 0; (* Флаг необходимости инициализации структур-дескрипторов *)

(* Модуль A1-15 *)
stDO_Ini(data_Ini := true, imit:=FALSE, strDO := od.do_0);
inits := inits + BOOL_TO_UINT(stDO_Ini.Init);

(* Модуль A1-16 *)
stDO_Ini(data_Ini := true, imit:=FALSE, strDO := od.do_1);
inits := inits + BOOL_TO_UINT(stDO_Ini.Init);

(* Модуль A1-17 *)
stDO_Ini(data_Ini := true, imit:=FALSE, strDO := od.do_2);
inits := inits + BOOL_TO_UINT(stDO_Ini.Init);

(* Модуль A1-18 *)
stDO_Ini(data_Ini := true, imit:=FALSE, strDO := od.do_3);
inits := inits + BOOL_TO_UINT(stDO_Ini.Init);

(* Модуль A1-19 *)
stDO_Ini(data_Ini := true, imit:=FALSE, strDO := od.do_4);
inits := inits + BOOL_TO_UINT(stDO_Ini.Init);

(* Модуль A1-23 *)
stDO_Ini(data_Ini := true, imit:=FALSE, strDO := od.gpio_out);
inits := inits + BOOL_TO_UINT(stDO_Ini.Init);
initiales := 0;

IF init THEN initiales := inits; END_IF;

(* ---- proc_IM.st ---- *)
FUNCTION_BLOCK proc_IM

VAR
	fb_Kran1 : fb_Kran; (*[A1-14:1, AI0] Резерв*)
	fb_Kran2 : fb_Kran; (*[A1-14:2, AI1] Резерв*)
	fb_Kran3 : fb_Kran;
	fb_Kran3b : fb_Kran;
	fb_Kran4 : fb_Kran;
	fb_Kran5 : fb_Kran;
	fb_Kran6 : fb_Kran;
	fb_nu1 : fb_OilPump;
	fb_nu2 : fb_OilPump;
	fb_pns : fb_Switch;
	fb_v1_Avom : fb_Switch;
	fb_v2_Avom : fb_Switch;
	fb_v3_Avom : fb_Switch;
	fb_v4_Avom : fb_Switch;
	fb_TEN_kollectora : fb_Switch;
	fb_KaloriferAVOM : fb_Switch;
	fb_CMN : fb_Switch;
	fb_TEN_MB : fb_Switch;
	fb_mv : fb_SectionSwitch;
	fb_PLC_Control : fb_meandr;
END_VAR

VAR_EXTERNAL
	di : DiConfig;
	od : DOconfig;
	IM : ImConfig;
END_VAR

VAR
	fb_dP_maslo_gaz_Less100 : fb_singleSignal;
	fb_dp_kran1_Less100 : fb_singleSignal;
	fb_QF1_on : fb_singleSignal;
	fb_QF2_on : fb_singleSignal;
	fb_QF23_on : fb_singleSignal;
	fb_QF4_QF5_on : fb_singleSignal;
	fb_QF6_QF7_on : fb_singleSignal;
	fb_QF8_QF9_on : fb_singleSignal;
	fb_QF10_QF11_on : fb_singleSignal;
	fb_QF12_QF13_on : fb_singleSignal;
	fb_QF14_QF15_on : fb_singleSignal;
	fb_QF22_on : fb_singleSignal;
	fb_NS_G1_G2 : fb_singleSignal;
	fb_NS_G3_G4 : fb_singleSignal;
	fb_NS_G15_G16 : fb_singleSignal;
	fb_NS_G17 : fb_singleSignal;
	fb_NS_G5_G6 : fb_singleSignal;
	fb_NS_G7_G8 : fb_singleSignal;
	fb_NS_G18_G19 : fb_singleSignal;
	fb_NS_G10_G11 : fb_singleSignal;
	fb_NS_G13_G14 : fb_singleSignal;
	fb_Vozbud_neispr_tsepey_upr_AVR_pit : fb_singleSignal;
	fb_Vozbud_gotovnost : fb_singleSignal;
	fb_Vozbud_neispravnost : fb_singleSignal;
	fb_SHAVR1_v_rabote : fb_singleSignal;
	fb_SHAVR2_v_rabote : fb_singleSignal;
	fb_Avariinoe_otkluch_vikluchatelya : fb_singleSignal;
	fb_Assinhronnii_hod_peregruzka : fb_singleSignal;
	fb_SHU_v_GPA_vkluch : fb_singleSignal;
	fb_SHP_v_GPA_vkluch : fb_singleSignal;
	fb_Uroven_masla_akkum : fb_singleSignal;
	fb_NKU1_GPA_on : fb_singleSignal;
	fb_NKU2_GPA_on : fb_singleSignal;
	fb_AO_KC_ot_SHKS : fb_singleSignal;
	fb_AO_GPA_ot_SHU : fb_singleSignal;
	fb_BEAO_srabotal : fb_singleSignal;
	fb_Chastotny_pusk : fb_singleSignal;
	fb_Neuspesh_chastotny_pusk : fb_singleSignal;
	fb_Rezhim_ruchnogo_regulirovaniya : fb_singleSignal;
	fb_Razreshenie_zagruzki_dvig : fb_singleSignal;
	fb_Osnovnoy_regul_off : fb_singleSignal;
	fb_Voltage_sekcii_norm : fb_singleSignal;
	fb_Reactorny_pusk : fb_singleSignal;
	fb_NO_GPA_ot_SHU : fb_singleSignal;
	fb_AO_GPA_ot_PRU : fb_singleSignal;
	fb_Nalichie_BP1 : fb_singleSignal;
	fb_Nalichie_BP2 : fb_singleSignal;
	fb_Nalichie_BP3 : fb_singleSignal;
	fb_Nalichie_BP4 : fb_singleSignal;
	fb_Nalichie_BP5 : fb_singleSignal;
	fb_Nalichie_BP6 : fb_singleSignal;
	fb_Nalichie_BP7_BP8 : fb_singleSignal;
	fb_Nalichie_BP9_BP10 : fb_singleSignal;
	fb_Nalichie_cepei_upravlen_mv : fb_singleSignal;
	fb_Nalichie_220BEAO : fb_singleSignal;
	fb_Nalichie_per_220_na_vhode : fb_singleSignal;
	fb_Nalichie_post_220_na_vhode : fb_singleSignal;
	fb_Nalichie_BP11 : fb_singleSignal;
	fb_Nalichie_BP12 : fb_singleSignal;
	fb_Dver_SHU_pered_otkrita : fb_singleSignal;
	fb_Dver_SHU_zad_otkrita : fb_singleSignal;
	fb_EO_GPA_ot_knopki_SHU : fb_singleSignal;
	fb_EO_EGPA_ot_PRY : fb_singleSignal;
	fb_Synchroniz_rezhima_K1 : fb_singleSignal;
	fb_Potok_ms_posle_AVOM : fb_singleSignal;
	fb_Avary_EGPA : fb_singleOutput;
	fb_U_lamp_SHU : fb_singleOutput;
	fb_AO_knopka_ind : fb_singleOutput;
	fb_Pusk : fb_singleOutput;
	fb_Stop_SHUP : fb_singleOutput;
	fb_NO_fonar : fb_singleOutput;
	fb_PC_fonar : fb_singleOutput;
	fb_AC_fonar : fb_singleOutput;
	fb_Kr1_smazka : fb_singleOutput;
	fb_Kr2_smazka : fb_singleOutput;
	fb_Kr4_open_from_alg : fb_singleOutput;
	fb_Synch_rej_K1 : fb_singleOutput;
	fb_Rabota_EGPA : fb_singleOutput;
	fb_Neispr_EGPA : fb_singleOutput;
END_VAR

(* Циклический опрос. ИМ *)

(* GPIO *)
fb_PLC_Control(output:=od.gpio_out.bits[0]);

(* Кран 1 *)
fb_Kran1(statOn := di.di_20.bits[5]._inversed,
         statOff := di.di_20.bits[4]._inversed,
         inSo := di.di_16.bits[0], inSz := di.di_16.bits[1],
         cmdOn:=od.do_0.bits[0], cmdOff:=od.do_0.bits[1],
         strKr:= IM.Kran1  );

(* Кран 2 *)
fb_Kran2(statOn := di.di_21.bits[0]._inversed,
         statOff := di.di_20.bits[7]._inversed,
         inSo := di.di_16.bits[2], inSz := di.di_16.bits[3],
         cmdOn:=od.do_0.bits[2], cmdOff:=od.do_0.bits[3],
         strKr:= IM.Kran2  );

(* Кран 3 *)
fb_Kran3(statOn := di.di_0.bits[5]._inversed,
         statOff := di.di_0.bits[4]._inversed,
         inSo := di.di_16.bits[4], inSz := di.di_16.bits[5],
         cmdOn:=od.do_0.bits[4], cmdOff:=od.do_0.bits[5],
         strKr:= IM.Kran3  );

(* Кран 3b *)
fb_Kran3b(statOn := di.di_0.bits[7]._inversed,
         statOff := di.di_0.bits[6]._inversed,
         inSo := di.di_16.bits[6], inSz := di.di_16.bits[7],
         cmdOn:=od.do_0.bits[6], cmdOff:=od.do_0.bits[7],
         strKr:= IM.Kran3b  );

(* Кран 4 *)
fb_Kran4(statOn := di.di_1.bits[1]._inversed,
         statOff := di.di_1.bits[0]._inversed,
         inSo := di.di_17.bits[0], inSz := di.di_17.bits[1],
         cmdOn:=od.do_0.bits[8], cmdOff:=od.do_0.bits[9],
         strKr:= IM.Kran4  );

(* Кран 5 *)
fb_Kran5(statOn := di.di_1.bits[3]._inversed,
         statOff := di.di_1.bits[2]._inversed,
         inSo := di.di_17.bits[2], inSz := di.di_17.bits[3],
         cmdOn:=od.do_0.bits[10], cmdOff:=od.do_0.bits[11],
         strKr:= IM.Kran5  );

(* Кран 6НР *)
fb_Kran6(statOn := di.di_1.bits[5]._inversed,
         statOff := di.di_1.bits[4]._inversed,
         inSo := di.di_17.bits[4], inSz := di.di_17.bits[5],
         cmdOn:=od.do_0.bits[12], cmdOff:=od.do_0.bits[13],
         strKr:= IM.Kran6  );

(*  НУ1 Насос уплотнения *)
fb_nu1(statOn := di.di_5.bits[1].value, statOff := di.di_5.bits[1]._inversed,
         cmdOn:=od.do_1.bits[4], cmdOff:=od.do_1.bits[5],
         StrSw:= IM.nu1  );

(*  НУ2 Насос уплотнения *)
fb_nu2(statOn := di.di_5.bits[2].value, statOff := di.di_5.bits[2]._inversed,
         cmdOn:=od.do_1.bits[6], cmdOff:=od.do_1.bits[7],
         StrSw:= IM.nu2  );

(*  ПНС Насос смазки *)
fb_pns(statOn := di.di_5.bits[0].value, statOff := di.di_5.bits[0]._inversed,
         cmdOn:=od.do_1.bits[0], cmdOff:=od.do_1.bits[1],
         StrSw:= IM.pns  );

(*  В1 АВОМ вентилятор охлаждения *)
fb_v1_Avom(statOn := di.di_5.bits[3].value, statOff := di.di_5.bits[3]._inversed,
         cmdOn:=od.do_1.bits[8], cmdOff:=od.do_1.bits[9],
         StrSw:= IM.v1_Avom  );

(*  В2 АВОМ вентилятор охлаждения *)
fb_v2_Avom(statOn := di.di_5.bits[4].value, statOff := di.di_5.bits[4]._inversed,
         cmdOn:=od.do_1.bits[10], cmdOff:=od.do_1.bits[11],
         StrSw:= IM.v2_Avom  );

(*  В3 АВОМ вентилятор охлаждения *)
fb_v3_Avom(statOn := di.di_5.bits[5].value, statOff := di.di_5.bits[5]._inversed,
         cmdOn:=od.do_1.bits[12], cmdOff:=od.do_1.bits[13],
         StrSw:= IM.v3_Avom  );

(*  В4 АВОМ вентилятор охлаждения *)
fb_v4_Avom(statOn := di.di_5.bits[6].value, statOff := di.di_5.bits[6]._inversed,
         cmdOn:=od.do_1.bits[14], cmdOff:=od.do_1.bits[15],
         StrSw:= IM.v4_Avom  );

(*  МВ масляный выключатель *)
fb_mv(statOn := di.di_7.bits[0].value, statOff := di.di_20.bits[3].value,
         basketRolledin:= di.di_7.bits[2], basketRolledout:= di.di_7.bits[2],
         cmdOn:=od.do_4.bits[6] , cmdOff:=od.do_4.bits[7],
         StrSw:= IM.mv  );

(* Тен коллектора *)
fb_TEN_kollectora(statOn := di.di_10.bits[1].value, statOff := di.di_10.bits[1]._inversed,
         cmdOn:=od.do_2.bits[6], cmdOff:=od.do_2.bits[6],
         StrSw:= IM.TEN_kollectora  );

(* Калорифер АВОМ *)
fb_KaloriferAVOM(statOn := di.di_10.bits[2].value, statOff := di.di_10.bits[2]._inversed,
         cmdOn:=od.do_2.bits[0], cmdOff:=od.do_2.bits[1],
         StrSw:= IM.KaloriferAVOM  );

(* ЦМН *)
fb_CMN(statOn := di.di_10.bits[3].value, statOff := di.di_10.bits[3]._inversed,
         cmdOn:=od.do_2.bits[4], cmdOff:=od.do_2.bits[5],
         StrSw:= IM.CMN);

(* Тен маслобака *)
fb_TEN_MB(statOn := di.di_10.bits[0].value, statOff := di.di_10.bits[0]._inversed,
         cmdOn:=od.do_2.bits[2], cmdOff:=od.do_2.bits[3],
         StrSw:= IM.TEN_MB);
(*************************************************** singleSignals ********************************************)

(* Перепад давления масло газ м*)
fb_dP_maslo_gaz_Less100(signal :=di.di_20.bits[6], str_SS := IM.SingleSignals.dP_maslo_gaz_Less100);

(* Перепад давления кран 1 *)
fb_dp_kran1_Less100(signal :=di.di_4.bits[1], str_SS := IM.SingleSignals.dp_kran1_Less100);

(* Неисправность цепей управления возбудителя *)
fb_Vozbud_neispr_tsepey_upr_AVR_pit(signal :=di.di_6.bits[4], str_SS := IM.SingleSignals.Vozbud_neispr_tsepey_upr_AVR_pit);

(* Возбудитель готовность *)
fb_Vozbud_gotovnost(signal :=di.di_6.bits[0], str_SS := IM.SingleSignals.Vozbud_gotovnost);

(* Возбудитель неисправность *)
fb_Vozbud_neispravnost(signal :=di.di_21.bits[7], str_SS := IM.SingleSignals.Vozbud_neispravnost);

(* ЩАВР 1 в работе *)
fb_SHAVR1_v_rabote(signal :=di.di_13.bits[6], str_SS := IM.SingleSignals.SHAVR1_v_rabote);

(* ЩАВР 2 в работе *)
fb_SHAVR2_v_rabote(signal :=di.di_13.bits[7], str_SS := IM.SingleSignals.SHAVR2_v_rabote);

(* ЩАВР 2 в работе *)
fb_Avariinoe_otkluch_vikluchatelya(signal :=di.di_8.bits[0], str_SS := IM.SingleSignals.Avariinoe_otkluch_vikluchatelya);

(* ЩАВР 2 в работе *)
fb_Assinhronnii_hod_peregruzka(signal :=di.di_8.bits[1], str_SS := IM.SingleSignals.Assinhronnii_hod_peregruzka);

(* ЩАВР 2 в работе *)
fb_SHU_v_GPA_vkluch(signal :=di.di_8.bits[2], str_SS := IM.SingleSignals.SHU_v_GPA_vkluch);

(* ЩАВР 2 в работе *)
fb_SHP_v_GPA_vkluch(signal :=di.di_8.bits[3], str_SS := IM.SingleSignals.SHP_v_GPA_vkluch);

(* ЩАВР 2 в работе *)
fb_Uroven_masla_akkum(signal :=di.di_4.bits[2], str_SS := IM.SingleSignals.Uroven_masla_akkum);

(* ЩАВР 2 в работе *)
fb_NKU1_GPA_on(signal :=di.di_10.bits[4], str_SS := IM.SingleSignals.NKU1_GPA_on);

(* ЩАВР 2 в работе *)
fb_NKU2_GPA_on(signal :=di.di_10.bits[5], str_SS := IM.SingleSignals.NKU2_GPA_on);

(* ЩАВР 2 в работе *)
fb_AO_KC_ot_SHKS(signal :=di.di_20.bits[0], str_SS := IM.SingleSignals.AO_KC_ot_SHKS);

(* ЩАВР 2 в работе *)
fb_AO_GPA_ot_SHU(signal :=di.di_21.bits[2], str_SS := IM.SingleSignals.AO_GPA_ot_SHU);

(* ЩАВР 2 в работе *)
fb_BEAO_srabotal(signal :=di.di_18.bits[1], str_SS := IM.SingleSignals.BEAO_srabotal);

(* ЩАВР 2 в работе *)
fb_Chastotny_pusk(signal :=di.di_9.bits[0], str_SS := IM.SingleSignals.Chastotny_pusk);

(* ЩАВР 2 в работе *)
fb_Neuspesh_chastotny_pusk(signal :=di.di_9.bits[1], str_SS := IM.SingleSignals.Neuspesh_chastotny_pusk);

(* ЩАВР 2 в работе *)
fb_Rezhim_ruchnogo_regulirovaniya(signal :=di.di_9.bits[2], str_SS := IM.SingleSignals.Rezhim_ruchnogo_regulirovaniya);

(* ЩАВР 2 в работе *)
fb_Razreshenie_zagruzki_dvig(signal :=di.di_6.bits[1], str_SS := IM.SingleSignals.Razreshenie_zagruzki_dvig);

(* ЩАВР 2 в работе *)
fb_Osnovnoy_regul_off(signal :=di.di_6.bits[3], str_SS := IM.SingleSignals.Osnovnoy_regul_off);

(* ЩАВР 2 в работе *)
fb_Voltage_sekcii_norm(signal :=di.di_8.bits[4], str_SS := IM.SingleSignals.Voltage_sekcii_norm);

(* ЩАВР 2 в работе *)
fb_Reactorny_pusk(signal :=di.di_8.bits[5], str_SS := IM.SingleSignals.Reactorny_pusk);

(* ЩАВР 2 в работе *)
fb_NO_GPA_ot_SHU(signal :=di.di_21.bits[1], str_SS := IM.SingleSignals.NO_GPA_ot_SHU);

(* ЩАВР 2 в работе *)
fb_AO_GPA_ot_PRU(signal :=di.di_21.bits[3], str_SS := IM.SingleSignals.AO_GPA_ot_PRU);

(* ЩАВР 2 в работе *)
fb_Nalichie_BP1(signal :=di.di_11.bits[0], str_SS := IM.SingleSignals.Nalichie_BP1);

(* ЩАВР 2 в работе *)
fb_Nalichie_BP2(signal :=di.di_11.bits[1], str_SS := IM.SingleSignals.Nalichie_BP2);

(* ЩАВР 2 в работе *)
fb_Nalichie_BP3(signal :=di.di_11.bits[2], str_SS := IM.SingleSignals.Nalichie_BP3);

(* ЩАВР 2 в работе *)
fb_Nalichie_BP4(signal :=di.di_11.bits[3], str_SS := IM.SingleSignals.Nalichie_BP4);

(* ЩАВР 2 в работе *)
fb_Nalichie_BP5(signal :=di.di_11.bits[4], str_SS := IM.SingleSignals.Nalichie_BP5);

(* ЩАВР 2 в работе *)
fb_Nalichie_BP6(signal :=di.di_11.bits[5], str_SS := IM.SingleSignals.Nalichie_BP6);

(* ЩАВР 2 в работе *)
fb_Nalichie_BP7_BP8(signal :=di.di_11.bits[6], str_SS := IM.SingleSignals.Nalichie_BP7_BP8);

(* ЩАВР 2 в работе *)
fb_Nalichie_BP9_BP10(signal :=di.di_11.bits[7], str_SS := IM.SingleSignals.Nalichie_BP9_BP10);

(* ЩАВР 2 в работе *)
fb_Nalichie_cepei_upravlen_mv(signal :=di.di_12.bits[0], str_SS := IM.SingleSignals.Nalichie_cepei_upravlen_mv);

(* ЩАВР 2 в работе *)
fb_Nalichie_220BEAO(signal :=di.di_12.bits[1], str_SS := IM.SingleSignals.Nalichie_220BEAO);

(* ЩАВР 2 в работе *)
fb_Nalichie_per_220_na_vhode(signal :=di.di_12.bits[2], str_SS := IM.SingleSignals.Nalichie_per_220_na_vhode);

(* ЩАВР 2 в работе *)
fb_Nalichie_post_220_na_vhode(signal :=di.di_12.bits[3], str_SS := IM.SingleSignals.Nalichie_post_220_na_vhode);

(* ЩАВР 2 в работе *)
fb_Nalichie_BP11(signal :=di.di_12.bits[4], str_SS := IM.SingleSignals.Nalichie_BP11);

(* ЩАВР 2 в работе *)
fb_Nalichie_BP12(signal :=di.di_12.bits[4], str_SS := IM.SingleSignals.Nalichie_BP12);

(* ЩАВР 2 в работе *)
fb_Dver_SHU_pered_otkrita(signal :=di.di_13.bits[0], str_SS := IM.SingleSignals.Dver_SHU_pered_otkrita);

(* ЩАВР 2 в работе *)
fb_Dver_SHU_zad_otkrita(signal :=di.di_13.bits[1], str_SS := IM.SingleSignals.Dver_SHU_zad_otkrita);

(* ЩАВР 2 в работе *)
fb_EO_GPA_ot_knopki_SHU(signal :=di.di_14.bits[0], str_SS := IM.SingleSignals.EO_GPA_ot_knopki_SHU);

(* ЩАВР 2 в работе *)
fb_EO_EGPA_ot_PRY(signal :=di.di_14.bits[1], str_SS := IM.SingleSignals.EO_EGPA_ot_PRY);

(* ЩАВР 2 в работе *)
fb_Synchroniz_rezhima_K1(signal :=di.di_3.bits[4], str_SS := IM.SingleSignals.Synchroniz_rezhima_K1);

(* ЩАВР 2 в работе *)
fb_Potok_ms_posle_AVOM(signal :=di.di_3.bits[4], str_SS := IM.SingleSignals.Potok_ms_posle_AVOM);

  (* Выключатель основного ввода питания QF1  в положении включен   *)
fb_QF1_on(signal :=di.di_7.bits[6], str_SS := IM.SingleSignals.QF1_on);

  (* Выключатель резервного ввода питания QF2  в положении включен   *)
fb_QF2_on(signal :=di.di_7.bits[7], str_SS := IM.SingleSignals.QF2_on);

  (* Выключатель питания кранов:  QF23 110 В в положении включен   *)
fb_QF23_on(signal :=di.di_8.bits[0], str_SS := IM.SingleSignals.QF23_on);

  (* Выключатели группы 1: QF4, QF5 в положении включен   *)
fb_QF4_QF5_on(signal :=di.di_8.bits[1], str_SS := IM.SingleSignals.QF4_QF5_on);

  (* Выключатели группы 2: QF6, QF7 в положении включен   *)
fb_QF6_QF7_on(signal :=di.di_8.bits[2], str_SS := IM.SingleSignals.QF6_QF7_on);

  (* Выключатели группы 3: QF8, QF9 в положении включен   *)
fb_QF8_QF9_on(signal :=di.di_8.bits[3], str_SS := IM.SingleSignals.QF8_QF9_on);

  (* Выключатели группы 4: QF10, QF11 в положении включен   *)
fb_QF10_QF11_on(signal :=di.di_8.bits[4], str_SS := IM.SingleSignals.QF10_QF11_on);

  (* Выключатели группы 5: QF12, QF13 в положении включен   *)
fb_QF12_QF13_on(signal :=di.di_8.bits[5], str_SS := IM.SingleSignals.QF12_QF13_on);

  (* Выключатели группы 6: QF14, QF15 в положении включен   *)
fb_QF14_QF15_on(signal :=di.di_8.bits[6], str_SS := IM.SingleSignals.QF14_QF15_on);

  (* Выключатели группы : QF22 в положении включен   *)
fb_QF22_on(signal :=di.di_14.bits[2], str_SS := IM.SingleSignals.QF22_on);

  (* Неисправность источников питания группы 1: G1, G2 (=24 В)   *)
fb_NS_G1_G2(signal :=di.di_8.bits[7], str_SS := IM.SingleSignals.NS_G1_G2);

  (* Неисправность источников питания группы 2: G3, G4 (=24 В)   *)
fb_NS_G3_G4(signal :=di.di_9.bits[0], str_SS := IM.SingleSignals.NS_G3_G4);

  (* Неисправность источников питания внутренних ПТС: G15, G16 (=24 В)   *)
fb_NS_G15_G16(signal :=di.di_9.bits[1], str_SS := IM.SingleSignals.NS_G15_G16);

  (* Неисправность источника питания аналоговых сигналов: G17 (=24 В)   *)
fb_NS_G17(signal :=di.di_9.bits[2], str_SS := IM.SingleSignals.NS_G17);

  (* Неисправность источников питания группы 3: G5, G6 (=24 В)   *)
fb_NS_G5_G6(signal :=di.di_9.bits[3], str_SS := IM.SingleSignals.NS_G5_G6);

  (* Неисправность источников питания группы 4: G7, G8 (=24 В)   *)
fb_NS_G7_G8(signal :=di.di_9.bits[4], str_SS := IM.SingleSignals.NS_G7_G8);

  (* Неисправность источников питания внешних цепей: G18, G19 (=24 В)   *)
fb_NS_G18_G19(signal :=di.di_9.bits[5], str_SS := IM.SingleSignals.NS_G18_G19);

  (* Неисправность источников питания группы 5: G9, G10, G11, G12 (=110 В)   *)
fb_NS_G10_G11(signal :=di.di_9.bits[6], str_SS := IM.SingleSignals.NS_G10_G11);

  (* Неисправность источников питания G13, G14 (=24 В)   *)
fb_NS_G13_G14(signal :=di.di_9.bits[7], str_SS := IM.SingleSignals.NS_G13_G14);

(*************************************************** SingleOutputs ********************************************)

(* Идикация НО (подсветка кнопки на шкафу)   *)
fb_Rabota_EGPA(str_SO := IM.SingleOutputs.Rabota_EGPA, signal:=od.do_4.bits[2]);

(* Взвод включения БЭАО по неисправности ПТС   *)
fb_Neispr_EGPA(str_SO := IM.SingleOutputs.Neispr_EGPA, signal:=od.do_4.bits[0]);

(* Авария ЭГПА в КЦ
fb_Avary_EGPA(str_SO := IM.SingleOutputs.Avary_EGPA, signal:=od.do_4.bits[1);  *)

(* Сброс включения БЭАО по неисправности ПТС   *)
fb_U_lamp_SHU(str_SO := IM.SingleOutputs.U_lamp_SHU, signal:=od.do_4.bits[3]);

(* Индикация ПС Фонарь   *)
fb_AO_knopka_ind(str_SO := IM.SingleOutputs.AO_knopka_ind, signal:=od.do_4.bits[4]);

(* Индикация АС Фонарь   *)
fb_Pusk(str_SO := IM.SingleOutputs.Pusk_SHUP, signal:=od.do_4.bits[8]);

(* Отключение МВ1 от КНА   *)
fb_Stop_SHUP(str_SO := IM.SingleOutputs.Stop_SHUP, signal:=od.do_4.bits[9]);

(* Отключение МВ1 от КНА   *)
fb_NO_fonar(str_SO := IM.SingleOutputs.NO_fonar, signal:=od.do_3.bits[10]);

(* Отключение МВ1 от КНА   *)
fb_PC_fonar(str_SO := IM.SingleOutputs.PC_fonar, signal:=od.do_3.bits[9]);

(* Отключение МВ1 от КНА   *)
fb_AC_fonar(str_SO := IM.SingleOutputs.AC_fonar, signal:=od.do_3.bits[8]);

(* Отключение МВ1 от КНА   *)
fb_Kr1_smazka(str_SO := IM.SingleOutputs.Kr1_smazka, signal:=od.do_0.bits[14]);

(* Отключение МВ1 от КНА   *)
fb_Kr2_smazka(str_SO := IM.SingleOutputs.Kr2_smazka, signal:=od.do_0.bits[15]);

(* Отключение МВ1 от КНА   *)
fb_Kr4_open_from_alg(str_SO := IM.SingleOutputs.Kr4_open_from_alg, signal:=od.do_0.bits[8]);

(* Отключение МВ1 от КНА   *)
fb_Synch_rej_K1(str_SO := IM.SingleOutputs.Synch_rej_K1, signal:=od.do_3.bits[13]);

 (**************************************** Аналоговые и Дискретные параметры ***********************************)
